Yaskawa INFORM job: A_ROOF_SIDE_0617_2_PAINT_48.JBI

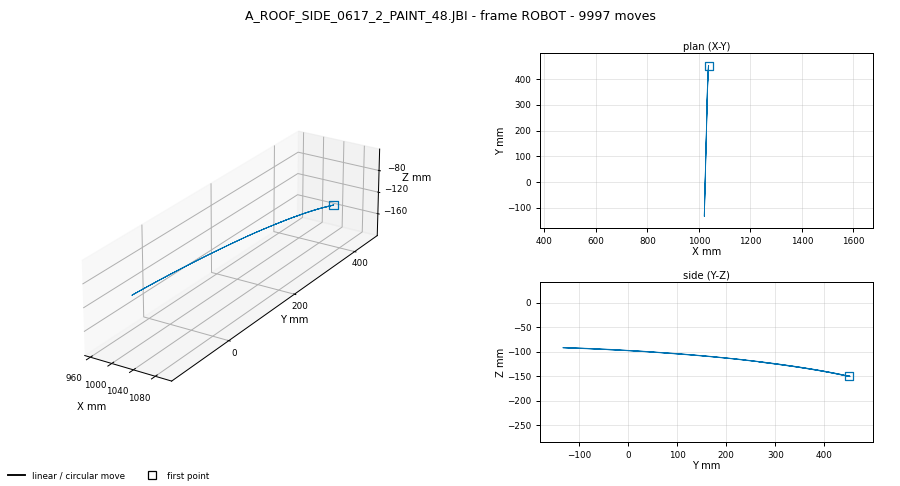
[picture p0: tool path of A_ROOF_SIDE_0617_2_PAINT_48.JBI in frame ROBOT, 9997 of 9997 moves have a stored position in this frame; points joined in program order, loops and branches not executed]
/JOB
//NAME A_ROOF_SIDE_0617_2_PAINT48
//POS
///NPOS 9997,0,0,0,0,0
///TOOL 1
///USER 0
///POSTYPE ROBOT
///RECTAN
///RCONF 1,0,0,0,0,0,0,0,0,0,0,0,0,0,0,0,0,0,0,0,0,0,0,0
C00000=1038.154,450.704,-149.023,176.566,47.258,159.897
C00001=1038.195,451.062,-149.082,176.595,47.266,159.904
C00002=1038.238,451.419,-149.141,176.623,47.275,159.910
C00003=1038.282,451.776,-149.199,176.652,47.283,159.916
C00004=1038.327,452.132,-149.255,176.680,47.290,159.922
C00005=1038.035,452.185,-149.577,176.684,47.363,159.945
C00006=1037.991,451.842,-149.523,176.655,47.356,159.939
C00007=1037.948,451.499,-149.468,176.628,47.348,159.933
C00008=1037.908,451.156,-149.412,176.601,47.340,159.927
C00009=1037.867,450.813,-149.355,176.574,47.332,159.921
C00010=1037.838,450.567,-149.314,176.554,47.326,159.916
C00011=1037.811,450.322,-149.271,176.535,47.321,159.912
C00012=1037.784,450.077,-149.230,176.516,47.315,159.908
C00013=1037.757,449.831,-149.186,176.496,47.309,159.904
C00014=1037.732,449.587,-149.144,176.477,47.303,159.899
C00015=1037.706,449.342,-149.100,176.459,47.296,159.895
C00016=1037.680,449.096,-149.056,176.440,47.290,159.890
C00017=1037.656,448.852,-149.011,176.421,47.283,159.886
C00018=1037.633,448.606,-148.966,176.403,47.277,159.882
C00019=1037.610,448.361,-148.921,176.384,47.271,159.877
C00020=1037.587,448.117,-148.875,176.366,47.263,159.873
C00021=1037.564,447.872,-148.829,176.348,47.257,159.868
C00022=1037.543,447.628,-148.782,176.328,47.250,159.864
C00023=1037.522,447.383,-148.734,176.310,47.243,159.859
C00024=1037.502,447.140,-148.687,176.292,47.236,159.855
C00025=1037.481,446.895,-148.639,176.274,47.229,159.850
C00026=1037.462,446.651,-148.590,176.256,47.221,159.846
C00027=1037.443,446.407,-148.542,176.237,47.214,159.841
C00028=1037.425,446.162,-148.492,176.220,47.207,159.837
C00029=1037.407,445.919,-148.443,176.203,47.199,159.832
C00030=1037.390,445.675,-148.391,176.184,47.192,159.828
C00031=1037.373,445.431,-148.341,176.167,47.184,159.823
C00032=1037.357,445.188,-148.290,176.149,47.177,159.818
C00033=1037.342,444.944,-148.238,176.132,47.169,159.814
C00034=1037.327,444.701,-148.186,176.115,47.161,159.809
C00035=1037.312,444.457,-148.134,176.098,47.153,159.805
C00036=1037.298,444.215,-148.081,176.080,47.145,159.800
C00037=1037.284,443.972,-148.027,176.063,47.136,159.795
C00038=1037.271,443.728,-147.974,176.046,47.128,159.790
C00039=1037.258,443.484,-147.920,176.029,47.120,159.786
C00040=1037.244,443.240,-147.867,176.013,47.112,159.781
C00041=1037.231,442.997,-147.814,175.995,47.104,159.777
C00042=1037.217,442.752,-147.761,175.979,47.096,159.772
C00043=1037.204,442.508,-147.708,175.962,47.087,159.768
C00044=1037.191,442.264,-147.654,175.945,47.080,159.763
C00045=1037.178,442.020,-147.601,175.928,47.072,159.759
C00046=1037.164,441.776,-147.549,175.912,47.063,159.754
C00047=1037.151,441.533,-147.495,175.895,47.055,159.750
C00048=1037.138,441.288,-147.443,175.879,47.047,159.745
C00049=1037.125,441.044,-147.390,175.862,47.040,159.741
C00050=1037.112,440.801,-147.337,175.845,47.032,159.736
C00051=1037.099,440.556,-147.285,175.829,47.024,159.732
C00052=1037.086,440.312,-147.232,175.813,47.016,159.728
C00053=1037.073,440.068,-147.179,175.798,47.008,159.723
C00054=1037.060,439.824,-147.126,175.782,47.000,159.719
C00055=1037.047,439.580,-147.075,175.766,46.993,159.715
C00056=1037.034,439.336,-147.022,175.749,46.985,159.710
C00057=1037.021,439.091,-146.970,175.733,46.977,159.706
C00058=1037.009,438.847,-146.917,175.717,46.970,159.702
C00059=1036.996,438.603,-146.866,175.701,46.962,159.697
C00060=1036.983,438.358,-146.813,175.686,46.954,159.693
C00061=1036.971,438.114,-146.761,175.670,46.946,159.689
C00062=1036.957,437.872,-146.709,175.654,46.939,159.685
C00063=1036.945,437.628,-146.657,175.639,46.931,159.681
C00064=1036.932,437.385,-146.606,175.624,46.924,159.677
C00065=1036.920,437.142,-146.553,175.609,46.916,159.672
C00066=1036.907,436.899,-146.502,175.593,46.909,159.668
C00067=1036.894,436.655,-146.450,175.578,46.901,159.664
C00068=1036.882,436.413,-146.399,175.562,46.894,159.660
C00069=1036.869,436.169,-146.348,175.548,46.886,159.656
C00070=1036.857,435.924,-146.296,175.532,46.879,159.652
C00071=1036.844,435.680,-146.245,175.517,46.871,159.648
C00072=1036.832,435.436,-146.193,175.502,46.864,159.644
C00073=1036.820,435.191,-146.142,175.487,46.857,159.640
C00074=1036.807,434.947,-146.091,175.472,46.849,159.636
C00075=1036.795,434.702,-146.039,175.457,46.842,159.632
C00076=1036.782,434.458,-145.988,175.442,46.835,159.628
C00077=1036.770,434.213,-145.937,175.427,46.828,159.624
C00078=1036.758,433.969,-145.886,175.413,46.821,159.620
C00079=1036.745,433.725,-145.835,175.398,46.813,159.616
C00080=1036.733,433.480,-145.784,175.384,46.806,159.612
C00081=1036.721,433.235,-145.734,175.369,46.799,159.609
C00082=1036.708,432.991,-145.683,175.354,46.792,159.605
C00083=1036.696,432.747,-145.632,175.340,46.785,159.601
C00084=1036.684,432.502,-145.581,175.325,46.778,159.597
C00085=1036.672,432.257,-145.530,175.311,46.771,159.593
C00086=1036.655,431.927,-145.462,175.292,46.762,159.588
C00087=1036.639,431.598,-145.394,175.272,46.752,159.583
C00088=1036.623,431.268,-145.327,175.253,46.742,159.578
C00089=1036.607,430.938,-145.258,175.234,46.733,159.573
C00090=1036.594,430.693,-145.208,175.220,46.726,159.569
C00091=1036.583,430.449,-145.158,175.207,46.719,159.566
C00092=1036.571,430.205,-145.107,175.193,46.712,159.562
C00093=1036.559,429.960,-145.057,175.178,46.706,159.558
C00094=1036.548,429.715,-145.006,175.164,46.699,159.555
C00095=1036.535,429.470,-144.956,175.151,46.692,159.551
C00096=1036.524,429.226,-144.906,175.137,46.685,159.547
C00097=1036.512,428.981,-144.856,175.123,46.678,159.544
C00098=1036.500,428.736,-144.806,175.110,46.671,159.540
C00099=1036.489,428.491,-144.756,175.096,46.665,159.537
C00100=1036.477,428.247,-144.706,175.083,46.658,159.533
C00101=1036.465,428.002,-144.657,175.069,46.651,159.529
C00102=1036.454,427.757,-144.607,175.055,46.645,159.526
C00103=1036.442,427.512,-144.557,175.042,46.638,159.522
C00104=1036.431,427.268,-144.508,175.028,46.631,159.519
C00105=1036.419,427.022,-144.458,175.015,46.625,159.515
C00106=1036.407,426.778,-144.409,175.002,46.618,159.512
C00107=1036.395,426.533,-144.359,174.988,46.612,159.509
C00108=1036.383,426.288,-144.310,174.976,46.605,159.505
C00109=1036.373,426.043,-144.260,174.962,46.599,159.502
C00110=1036.361,425.798,-144.211,174.949,46.592,159.498
C00111=1036.349,425.553,-144.162,174.936,46.586,159.495
C00112=1036.338,425.308,-144.113,174.922,46.579,159.491
C00113=1036.327,425.063,-144.064,174.910,46.573,159.488
C00114=1036.315,424.819,-144.015,174.897,46.566,159.485
C00115=1036.304,424.574,-143.966,174.884,46.560,159.481
C00116=1036.292,424.329,-143.917,174.871,46.554,159.478
C00117=1036.281,424.084,-143.868,174.858,46.548,159.475
C00118=1036.270,423.839,-143.818,174.845,46.541,159.471
C00119=1036.259,423.595,-143.769,174.833,46.535,159.468
C00120=1036.247,423.348,-143.721,174.820,46.528,159.465
C00121=1036.235,423.104,-143.672,174.807,46.522,159.461
C00122=1036.218,422.706,-143.593,174.787,46.512,159.456
C00123=1036.199,422.308,-143.515,174.767,46.502,159.451
C00124=1036.181,421.909,-143.436,174.747,46.492,159.446
C00125=1036.163,421.511,-143.357,174.726,46.482,159.441
C00126=1036.151,421.265,-143.309,174.714,46.476,159.437
C00127=1036.140,421.021,-143.261,174.702,46.470,159.434
C00128=1036.129,420.776,-143.212,174.689,46.464,159.431
C00129=1036.118,420.531,-143.164,174.677,46.458,159.428
C00130=1036.107,420.286,-143.116,174.664,46.452,159.425
C00131=1036.096,420.041,-143.068,174.653,46.446,159.422
C00132=1036.085,419.796,-143.020,174.641,46.440,159.419
C00133=1036.074,419.550,-142.971,174.628,46.434,159.416
C00134=1036.063,419.305,-142.925,174.616,46.428,159.413
C00135=1036.052,419.060,-142.876,174.604,46.423,159.410
C00136=1036.041,418.815,-142.828,174.593,46.417,159.407
C00137=1036.030,418.570,-142.780,174.580,46.411,159.403
C00138=1036.020,418.324,-142.733,174.568,46.405,159.400
C00139=1036.009,418.079,-142.685,174.557,46.399,159.397
C00140=1035.998,417.834,-142.636,174.545,46.393,159.394
C00141=1035.987,417.589,-142.590,174.533,46.388,159.391
C00142=1035.977,417.344,-142.542,174.521,46.382,159.388
C00143=1035.966,417.098,-142.494,174.509,46.376,159.385
C00144=1035.955,416.852,-142.447,174.498,46.370,159.383
C00145=1035.944,416.608,-142.399,174.486,46.365,159.380
C00146=1035.933,416.363,-142.352,174.475,46.359,159.377
C00147=1035.922,416.117,-142.305,174.463,46.353,159.374
C00148=1035.912,415.872,-142.258,174.452,46.348,159.371
C00149=1035.901,415.626,-142.210,174.440,46.342,159.368
C00150=1035.890,415.381,-142.164,174.429,46.337,159.365
C00151=1035.880,415.136,-142.116,174.417,46.331,159.362
C00152=1035.869,414.891,-142.069,174.406,46.325,159.359
C00153=1035.858,414.644,-142.022,174.394,46.320,159.357
C00154=1035.847,414.399,-141.976,174.383,46.314,159.354
C00155=1035.837,414.154,-141.928,174.372,46.309,159.351
C00156=1035.827,413.909,-141.881,174.360,46.303,159.348
C00157=1035.816,413.664,-141.835,174.349,46.298,159.345
C00158=1035.806,413.419,-141.787,174.339,46.292,159.342
C00159=1035.794,413.172,-141.741,174.327,46.287,159.340
C00160=1035.784,412.927,-141.694,174.316,46.281,159.337
C00161=1035.773,412.682,-141.647,174.305,46.276,159.334
C00162=1035.763,412.436,-141.601,174.294,46.271,159.331
C00163=1035.753,412.191,-141.554,174.282,46.265,159.329
C00164=1035.742,411.946,-141.507,174.272,46.260,159.326
C00165=1035.732,411.700,-141.460,174.261,46.254,159.323
C00166=1035.722,411.455,-141.415,174.250,46.249,159.320
C00167=1035.712,411.210,-141.368,174.239,46.244,159.318
C00168=1035.702,410.964,-141.322,174.229,46.239,159.315
C00169=1035.691,410.719,-141.276,174.218,46.233,159.312
C00170=1035.681,410.473,-141.229,174.206,46.228,159.310
C00171=1035.670,410.228,-141.183,174.196,46.223,159.307
C00172=1035.660,409.982,-141.137,174.185,46.218,159.304
C00173=1035.649,409.737,-141.091,174.174,46.213,159.302
C00174=1035.639,409.491,-141.044,174.164,46.208,159.299
C00175=1035.628,409.245,-140.998,174.153,46.203,159.297
C00176=1035.618,409.000,-140.953,174.143,46.197,159.294
C00177=1035.608,408.755,-140.907,174.132,46.192,159.291
C00178=1035.598,408.517,-140.863,174.122,46.188,159.289
C00179=1035.588,408.280,-140.819,174.112,46.182,159.286
C00180=1035.578,408.043,-140.775,174.102,46.177,159.284
C00181=1035.569,407.805,-140.730,174.091,46.173,159.281
C00182=1035.559,407.568,-140.686,174.082,46.168,159.279
C00183=1035.549,407.330,-140.642,174.072,46.163,159.277
C00184=1035.539,407.093,-140.598,174.061,46.159,159.274
C00185=1035.530,406.855,-140.554,174.052,46.153,159.272
C00186=1035.519,406.610,-140.508,174.041,46.148,159.269
C00187=1035.510,406.365,-140.462,174.031,46.144,159.267
C00188=1035.499,406.118,-140.417,174.021,46.139,159.264
C00189=1035.489,405.874,-140.371,174.010,46.134,159.262
C00190=1035.479,405.627,-140.326,174.001,46.129,159.259
C00191=1035.469,405.382,-140.281,173.990,46.124,159.257
C00192=1035.460,405.136,-140.235,173.980,46.119,159.254
C00193=1035.450,404.890,-140.190,173.970,46.114,159.252
C00194=1035.440,404.645,-140.145,173.960,46.110,159.249
C00195=1035.429,404.399,-140.099,173.950,46.104,159.247
C00196=1035.420,404.154,-140.054,173.940,46.100,159.244
C00197=1035.411,403.908,-140.009,173.929,46.095,159.242
C00198=1035.400,403.662,-139.964,173.920,46.090,159.240
C00199=1035.391,403.416,-139.919,173.910,46.086,159.237
C00200=1035.381,403.171,-139.873,173.900,46.081,159.235
C00201=1035.371,402.926,-139.828,173.890,46.076,159.233
C00202=1035.361,402.679,-139.783,173.880,46.072,159.230
C00203=1035.352,402.433,-139.739,173.871,46.067,159.228
C00204=1035.342,402.188,-139.694,173.861,46.062,159.225
C00205=1035.333,401.942,-139.649,173.851,46.058,159.223
C00206=1035.323,401.697,-139.604,173.841,46.053,159.221
C00207=1035.313,401.450,-139.559,173.831,46.049,159.218
C00208=1035.303,401.205,-139.514,173.822,46.044,159.216
C00209=1035.293,400.959,-139.470,173.812,46.039,159.214
C00210=1035.284,400.713,-139.425,173.802,46.034,159.211
C00211=1035.274,400.468,-139.380,173.792,46.030,159.209
C00212=1035.264,400.222,-139.337,173.783,46.026,159.207
C00213=1035.254,399.976,-139.292,173.773,46.021,159.205
C00214=1035.245,399.730,-139.248,173.764,46.017,159.202
C00215=1035.235,399.485,-139.203,173.755,46.012,159.200
C00216=1035.226,399.239,-139.159,173.745,46.008,159.198
C00217=1035.216,398.993,-139.114,173.736,46.003,159.196
C00218=1035.207,398.747,-139.070,173.726,45.999,159.193
C00219=1035.196,398.501,-139.026,173.717,45.994,159.191
C00220=1035.187,398.255,-138.982,173.707,45.990,159.189
C00221=1035.177,398.010,-138.938,173.698,45.986,159.187
C00222=1035.168,397.764,-138.894,173.689,45.981,159.185
C00223=1035.158,397.518,-138.850,173.679,45.977,159.182
C00224=1035.149,397.272,-138.806,173.670,45.973,159.180
C00225=1035.139,397.026,-138.762,173.661,45.969,159.178
C00226=1035.130,396.780,-138.718,173.651,45.964,159.176
C00227=1035.120,396.535,-138.675,173.642,45.960,159.174
C00228=1035.111,396.289,-138.631,173.633,45.956,159.172
C00229=1035.102,396.042,-138.587,173.624,45.951,159.169
C00230=1035.092,395.796,-138.542,173.614,45.947,159.167
C00231=1035.083,395.551,-138.499,173.605,45.943,159.165
C00232=1035.073,395.305,-138.455,173.596,45.939,159.163
C00233=1035.064,395.059,-138.411,173.588,45.934,159.161
C00234=1035.055,394.814,-138.367,173.578,45.930,159.159
C00235=1035.045,394.568,-138.324,173.569,45.927,159.157
C00236=1035.036,394.321,-138.280,173.560,45.922,159.155
C00237=1035.026,394.076,-138.237,173.551,45.918,159.153
C00238=1035.018,393.848,-138.196,173.543,45.914,159.151
C00239=1035.010,393.621,-138.157,173.535,45.910,159.149
C00240=1035.001,393.394,-138.117,173.527,45.907,159.147
C00241=1034.992,393.167,-138.077,173.518,45.903,159.145
C00242=1034.983,392.940,-138.037,173.510,45.899,159.143
C00243=1034.976,392.712,-137.997,173.502,45.896,159.141
C00244=1034.966,392.485,-137.957,173.493,45.892,159.139
C00245=1034.958,392.258,-137.917,173.486,45.888,159.138
C00246=1034.948,392.012,-137.874,173.477,45.884,159.135
C00247=1034.940,391.766,-137.831,173.467,45.880,159.133
C00248=1034.930,391.520,-137.787,173.459,45.877,159.132
C00249=1034.921,391.274,-137.744,173.450,45.872,159.129
C00250=1034.912,391.028,-137.701,173.441,45.869,159.127
C00251=1034.903,390.782,-137.659,173.433,45.865,159.126
C00252=1034.894,390.536,-137.615,173.424,45.861,159.123
C00253=1034.884,390.290,-137.572,173.415,45.857,159.122
C00254=1034.875,390.044,-137.529,173.407,45.853,159.120
C00255=1034.866,389.798,-137.487,173.398,45.849,159.118
C00256=1034.856,389.551,-137.444,173.390,45.846,159.116
C00257=1034.848,389.305,-137.401,173.381,45.841,159.114
C00258=1034.839,389.060,-137.358,173.373,45.837,159.112
C00259=1034.829,388.814,-137.316,173.365,45.833,159.110
C00260=1034.821,388.567,-137.273,173.356,45.830,159.108
C00261=1034.811,388.321,-137.231,173.347,45.826,159.106
C00262=1034.803,388.075,-137.188,173.339,45.822,159.104
C00263=1034.794,387.829,-137.145,173.331,45.819,159.102
C00264=1034.784,387.583,-137.103,173.322,45.815,159.100
C00265=1034.776,387.336,-137.060,173.313,45.812,159.099
C00266=1034.766,387.090,-137.018,173.305,45.808,159.097
C00267=1034.757,386.844,-136.975,173.297,45.804,159.095
C00268=1034.748,386.598,-136.934,173.289,45.801,159.093
C00269=1034.739,386.352,-136.891,173.280,45.797,159.091
C00270=1034.729,386.105,-136.849,173.272,45.793,159.089
C00271=1034.720,385.860,-136.807,173.264,45.790,159.087
C00272=1034.712,385.613,-136.764,173.255,45.786,159.086
C00273=1034.703,385.366,-136.723,173.248,45.783,159.084
C00274=1034.694,385.121,-136.680,173.239,45.779,159.082
C00275=1034.685,384.874,-136.638,173.231,45.776,159.080
C00276=1034.676,384.628,-136.597,173.222,45.772,159.078
C00277=1034.667,384.382,-136.554,173.214,45.769,159.077
C00278=1034.658,384.136,-136.513,173.206,45.765,159.075
C00279=1034.649,383.890,-136.471,173.198,45.761,159.073
C00280=1034.641,383.643,-136.429,173.190,45.758,159.071
C00281=1034.631,383.397,-136.386,173.182,45.754,159.069
C00282=1034.622,383.151,-136.344,173.174,45.751,159.068
C00283=1034.614,382.904,-136.303,173.166,45.748,159.066
C00284=1034.605,382.658,-136.261,173.158,45.744,159.064
C00285=1034.596,382.412,-136.219,173.150,45.740,159.062
C00286=1034.587,382.166,-136.178,173.142,45.737,159.061
C00287=1034.578,381.920,-136.136,173.134,45.734,159.059
C00288=1034.569,381.673,-136.094,173.126,45.730,159.057
C00289=1034.561,381.427,-136.053,173.118,45.727,159.055
C00290=1034.552,381.180,-136.010,173.110,45.723,159.054
C00291=1034.543,380.934,-135.969,173.102,45.720,159.052
C00292=1034.535,380.688,-135.928,173.095,45.716,159.050
C00293=1034.526,380.441,-135.886,173.087,45.713,159.048
C00294=1034.518,380.195,-135.845,173.078,45.710,159.047
C00295=1034.509,379.948,-135.803,173.071,45.707,159.045
C00296=1034.500,379.703,-135.762,173.063,45.703,159.043
C00297=1034.492,379.456,-135.721,173.055,45.700,159.042
C00298=1034.484,379.246,-135.685,173.049,45.698,159.040
C00299=1034.477,379.037,-135.650,173.042,45.695,159.039
C00300=1034.470,378.826,-135.614,173.036,45.691,159.037
C00301=1034.463,378.617,-135.580,173.029,45.689,159.036
C00302=1034.455,378.407,-135.544,173.022,45.686,159.035
C00303=1034.448,378.198,-135.509,173.016,45.683,159.033
C00304=1034.441,377.988,-135.474,173.009,45.681,159.032
C00305=1034.434,377.778,-135.440,173.002,45.678,159.030
C00306=1034.425,377.532,-135.398,172.996,45.675,159.029
C00307=1034.416,377.285,-135.357,172.987,45.672,159.027
C00308=1034.408,377.038,-135.316,172.980,45.669,159.026
C00309=1034.398,376.792,-135.275,172.972,45.666,159.024
C00310=1034.390,376.545,-135.234,172.965,45.663,159.022
C00311=1034.382,376.299,-135.194,172.957,45.659,159.021
C00312=1034.373,376.052,-135.153,172.950,45.657,159.019
C00313=1034.364,375.806,-135.112,172.943,45.653,159.018
C00314=1034.355,375.560,-135.071,172.935,45.650,159.016
C00315=1034.347,375.313,-135.030,172.927,45.647,159.014
C00316=1034.339,375.066,-134.989,172.919,45.644,159.013
C00317=1034.330,374.820,-134.949,172.912,45.641,159.011
C00318=1034.321,374.573,-134.908,172.905,45.638,159.010
C00319=1034.313,374.327,-134.867,172.897,45.635,159.008
C00320=1034.305,374.080,-134.826,172.890,45.632,159.007
C00321=1034.296,373.834,-134.786,172.882,45.629,159.005
C00322=1034.288,373.588,-134.746,172.875,45.626,159.003
C00323=1034.279,373.341,-134.705,172.868,45.623,159.002
C00324=1034.270,373.095,-134.665,172.860,45.620,159.000
C00325=1034.262,372.849,-134.624,172.853,45.617,158.999
C00326=1034.254,372.601,-134.584,172.846,45.614,158.997
C00327=1034.246,372.355,-134.543,172.839,45.612,158.996
C00328=1034.237,372.109,-134.503,172.831,45.609,158.994
C00329=1034.229,371.862,-134.462,172.824,45.606,158.993
C00330=1034.221,371.615,-134.422,172.817,45.603,158.991
C00331=1034.213,371.369,-134.382,172.810,45.600,158.990
C00332=1034.204,371.123,-134.342,172.802,45.597,158.988
C00333=1034.196,370.875,-134.301,172.795,45.594,158.987
C00334=1034.188,370.629,-134.261,172.788,45.591,158.985
C00335=1034.179,370.383,-134.221,172.781,45.588,158.984
C00336=1034.171,370.136,-134.181,172.773,45.586,158.982
C00337=1034.163,369.890,-134.140,172.766,45.583,158.981
C00338=1034.154,369.642,-134.100,172.759,45.580,158.979
C00339=1034.146,369.396,-134.060,172.753,45.577,158.978
C00340=1034.138,369.149,-134.020,172.746,45.575,158.977
C00341=1034.130,368.903,-133.980,172.738,45.572,158.975
C00342=1034.121,368.657,-133.940,172.731,45.569,158.974
C00343=1034.112,368.409,-133.901,172.724,45.567,158.972
C00344=1034.105,368.162,-133.861,172.717,45.564,158.971
C00345=1034.096,367.916,-133.822,172.711,45.561,158.970
C00346=1034.088,367.669,-133.782,172.703,45.559,158.968
C00347=1034.080,367.423,-133.742,172.696,45.556,158.967
C00348=1034.071,367.176,-133.702,172.689,45.553,158.965
C00349=1034.063,366.929,-133.662,172.682,45.550,158.964
C00350=1034.055,366.683,-133.623,172.675,45.548,158.962
C00351=1034.047,366.436,-133.583,172.668,45.545,158.961
C00352=1034.039,366.189,-133.544,172.662,45.543,158.960
C00353=1034.030,365.943,-133.504,172.655,45.540,158.958
C00354=1034.023,365.696,-133.464,172.648,45.537,158.957
C00355=1034.014,365.449,-133.425,172.640,45.535,158.956
C00356=1034.006,365.203,-133.386,172.633,45.532,158.954
C00357=1033.998,364.956,-133.346,172.627,45.530,158.953
C00358=1033.985,364.557,-133.283,172.616,45.526,158.951
C00359=1033.972,364.158,-133.219,172.605,45.522,158.948
C00360=1033.958,363.759,-133.155,172.594,45.518,158.946
C00361=1033.945,363.361,-133.092,172.584,45.514,158.944
C00362=1033.938,363.114,-133.052,172.577,45.511,158.943
C00363=1033.929,362.867,-133.013,172.570,45.508,158.941
C00364=1033.921,362.620,-132.974,172.563,45.506,158.940
C00365=1033.913,362.373,-132.934,172.557,45.503,158.939
C00366=1033.905,362.126,-132.895,172.550,45.501,158.938
C00367=1033.898,361.879,-132.856,172.543,45.499,158.936
C00368=1033.890,361.633,-132.817,172.537,45.496,158.935
C00369=1033.882,361.386,-132.778,172.530,45.494,158.934
C00370=1033.873,361.139,-132.739,172.523,45.492,158.932
C00371=1033.865,360.892,-132.700,172.517,45.489,158.931
C00372=1033.858,360.646,-132.660,172.510,45.487,158.930
C00373=1033.850,360.398,-132.622,172.503,45.484,158.928
C00374=1033.841,360.152,-132.583,172.497,45.482,158.927
C00375=1033.833,359.905,-132.544,172.490,45.480,158.926
C00376=1033.826,359.658,-132.506,172.483,45.477,158.925
C00377=1033.817,359.412,-132.466,172.478,45.475,158.923
C00378=1033.809,359.164,-132.428,172.471,45.473,158.922
C00379=1033.801,358.918,-132.390,172.465,45.470,158.921
C00380=1033.793,358.671,-132.351,172.458,45.468,158.920
C00381=1033.785,358.423,-132.312,172.451,45.466,158.918
C00382=1033.777,358.177,-132.273,172.445,45.464,158.917
C00383=1033.769,357.930,-132.235,172.438,45.461,158.916
C00384=1033.761,357.683,-132.196,172.432,45.459,158.915
C00385=1033.753,357.437,-132.158,172.425,45.457,158.913
C00386=1033.745,357.189,-132.119,172.419,45.454,158.912
C00387=1033.738,356.943,-132.081,172.413,45.453,158.911
C00388=1033.729,356.696,-132.042,172.406,45.450,158.910
C00389=1033.721,356.448,-132.004,172.400,45.448,158.909
C00390=1033.714,356.202,-131.966,172.393,45.446,158.907
C00391=1033.706,355.954,-131.926,172.388,45.443,158.906
C00392=1033.699,355.708,-131.888,172.381,45.442,158.905
C00393=1033.690,355.461,-131.850,172.375,45.440,158.904
C00394=1033.682,355.214,-131.812,172.368,45.437,158.903
C00395=1033.675,354.967,-131.774,172.362,45.436,158.902
C00396=1033.667,354.720,-131.736,172.356,45.433,158.900
C00397=1033.659,354.473,-131.697,172.350,45.431,158.899
C00398=1033.651,354.226,-131.659,172.343,45.429,158.898
C00399=1033.643,353.979,-131.622,172.337,45.427,158.897
C00400=1033.635,353.732,-131.583,172.330,45.425,158.896
C00401=1033.627,353.485,-131.545,172.325,45.423,158.895
C00402=1033.620,353.238,-131.507,172.318,45.420,158.893
C00403=1033.612,352.991,-131.469,172.312,45.419,158.892
C00404=1033.603,352.744,-131.431,172.306,45.417,158.891
C00405=1033.596,352.497,-131.393,172.300,45.415,158.890
C00406=1033.588,352.250,-131.355,172.293,45.412,158.889
C00407=1033.581,352.003,-131.317,172.287,45.411,158.888
C00408=1033.573,351.756,-131.279,172.282,45.408,158.886
C00409=1033.565,351.509,-131.241,172.275,45.407,158.885
C00410=1033.557,351.262,-131.203,172.269,45.405,158.884
C00411=1033.550,351.015,-131.166,172.264,45.403,158.883
C00412=1033.542,350.768,-131.127,172.257,45.401,158.882
C00413=1033.534,350.521,-131.090,172.251,45.399,158.881
C00414=1033.522,350.128,-131.030,172.242,45.396,158.879
C00415=1033.510,349.736,-130.970,172.231,45.393,158.877
C00416=1033.498,349.343,-130.910,172.222,45.390,158.876
C00417=1033.485,348.951,-130.850,172.213,45.387,158.874
C00418=1033.478,348.703,-130.813,172.207,45.385,158.873
C00419=1033.470,348.457,-130.776,172.200,45.383,158.872
C00420=1033.463,348.209,-130.738,172.195,45.381,158.871
C00421=1033.454,347.963,-130.700,172.188,45.379,158.870
C00422=1033.447,347.715,-130.663,172.182,45.377,158.868
C00423=1033.439,347.468,-130.625,172.177,45.376,158.868
C00424=1033.431,347.221,-130.588,172.171,45.374,158.866
C00425=1033.424,346.974,-130.551,172.165,45.372,158.865
C00426=1033.416,346.727,-130.514,172.159,45.370,158.864
C00427=1033.408,346.480,-130.476,172.153,45.369,158.863
C00428=1033.400,346.233,-130.439,172.147,45.367,158.862
C00429=1033.393,345.986,-130.402,172.141,45.365,158.861
C00430=1033.385,345.739,-130.365,172.136,45.363,158.860
C00431=1033.378,345.491,-130.328,172.129,45.362,158.859
C00432=1033.370,345.244,-130.291,172.124,45.359,158.858
C00433=1033.363,344.997,-130.253,172.118,45.358,158.857
C00434=1033.356,344.750,-130.216,172.113,45.356,158.856
C00435=1033.348,344.503,-130.179,172.106,45.354,158.855
C00436=1033.340,344.256,-130.142,172.101,45.353,158.854
C00437=1033.333,344.009,-130.105,172.095,45.351,158.853
C00438=1033.325,343.762,-130.068,172.089,45.350,158.852
C00439=1033.318,343.515,-130.031,172.083,45.348,158.851
C00440=1033.310,343.267,-129.994,172.077,45.346,158.850
C00441=1033.303,343.020,-129.957,172.072,45.344,158.849
C00442=1033.295,342.773,-129.920,172.066,45.343,158.848
C00443=1033.288,342.525,-129.883,172.060,45.341,158.847
C00444=1033.280,342.279,-129.846,172.054,45.340,158.846
C00445=1033.273,342.031,-129.809,172.049,45.338,158.845
C00446=1033.265,341.784,-129.773,172.044,45.336,158.844
C00447=1033.257,341.537,-129.736,172.038,45.335,158.843
C00448=1033.250,341.289,-129.699,172.032,45.333,158.842
C00449=1033.242,341.043,-129.662,172.026,45.331,158.841
C00450=1033.235,340.795,-129.625,172.021,45.329,158.840
C00451=1033.227,340.547,-129.589,172.015,45.328,158.839
C00452=1033.219,340.301,-129.552,172.009,45.327,158.838
C00453=1033.212,340.054,-129.516,172.003,45.325,158.837
C00454=1033.205,339.806,-129.480,171.998,45.323,158.836
C00455=1033.197,339.559,-129.442,171.992,45.322,158.835
C00456=1033.190,339.312,-129.406,171.987,45.321,158.834
C00457=1033.182,339.064,-129.370,171.982,45.319,158.834
C00458=1033.174,338.818,-129.333,171.976,45.318,158.833
C00459=1033.166,338.570,-129.297,171.970,45.316,158.832
C00460=1033.160,338.323,-129.260,171.964,45.315,158.831
C00461=1033.152,338.076,-129.224,171.959,45.313,158.830
C00462=1033.145,337.828,-129.188,171.953,45.312,158.829
C00463=1033.137,337.581,-129.152,171.948,45.310,158.828
C00464=1033.129,337.334,-129.115,171.943,45.309,158.827
C00465=1033.122,337.087,-129.079,171.937,45.307,158.826
C00466=1033.115,336.839,-129.042,171.931,45.306,158.825
C00467=1033.107,336.592,-129.006,171.926,45.304,158.824
C00468=1033.100,336.345,-128.970,171.920,45.303,158.823
C00469=1033.093,336.098,-128.934,171.915,45.302,158.823
C00470=1033.081,335.702,-128.875,171.907,45.300,158.821
C00471=1033.070,335.306,-128.818,171.898,45.297,158.820
C00472=1033.057,334.910,-128.760,171.889,45.295,158.818
C00473=1033.045,334.513,-128.702,171.880,45.293,158.817
C00474=1033.038,334.267,-128.666,171.875,45.291,158.816
C00475=1033.030,334.019,-128.630,171.869,45.290,158.815
C00476=1033.023,333.772,-128.594,171.864,45.289,158.814
C00477=1033.016,333.524,-128.559,171.859,45.287,158.813
C00478=1033.008,333.277,-128.523,171.853,45.287,158.812
C00479=1033.001,333.030,-128.487,171.848,45.285,158.812
C00480=1032.994,332.782,-128.451,171.843,45.284,158.811
C00481=1032.986,332.535,-128.415,171.838,45.282,158.810
C00482=1032.979,332.288,-128.379,171.832,45.281,158.809
C00483=1032.972,332.040,-128.344,171.827,45.280,158.808
C00484=1032.964,331.793,-128.308,171.822,45.278,158.807
C00485=1032.956,331.546,-128.272,171.816,45.278,158.807
C00486=1032.950,331.299,-128.237,171.811,45.276,158.806
C00487=1032.942,331.051,-128.201,171.806,45.275,158.805
C00488=1032.935,330.804,-128.166,171.801,45.274,158.804
C00489=1032.927,330.556,-128.129,171.795,45.272,158.803
C00490=1032.921,330.309,-128.094,171.790,45.271,158.802
C00491=1032.913,330.062,-128.058,171.785,45.270,158.802
C00492=1032.906,329.814,-128.023,171.780,45.269,158.801
C00493=1032.899,329.567,-127.987,171.774,45.268,158.800
C00494=1032.891,329.320,-127.952,171.769,45.266,158.799
C00495=1032.883,329.072,-127.916,171.764,45.265,158.798
C00496=1032.877,328.825,-127.881,171.759,45.264,158.797
C00497=1032.869,328.578,-127.845,171.753,45.263,158.797
C00498=1032.862,328.330,-127.810,171.748,45.262,158.796
C00499=1032.855,328.083,-127.774,171.743,45.261,158.795
C00500=1032.847,327.835,-127.739,171.738,45.259,158.794
C00501=1032.840,327.588,-127.704,171.733,45.258,158.793
C00502=1032.832,327.340,-127.669,171.727,45.258,158.793
C00503=1032.825,327.093,-127.634,171.722,45.256,158.792
C00504=1032.818,326.846,-127.599,171.717,45.255,158.791
C00505=1032.810,326.598,-127.564,171.713,45.254,158.790
C00506=1032.803,326.351,-127.529,171.706,45.253,158.789
C00507=1032.796,326.103,-127.493,171.702,45.252,158.789
C00508=1032.788,325.856,-127.459,171.697,45.251,158.788
C00509=1032.781,325.608,-127.424,171.692,45.250,158.787
C00510=1032.773,325.361,-127.389,171.687,45.249,158.786
C00511=1032.766,325.113,-127.354,171.681,45.248,158.786
C00512=1032.759,324.866,-127.319,171.676,45.247,158.785
C00513=1032.752,324.618,-127.284,171.671,45.246,158.784
C00514=1032.744,324.371,-127.249,171.667,45.245,158.784
C00515=1032.737,324.124,-127.214,171.662,45.245,158.783
C00516=1032.729,323.876,-127.179,171.657,45.243,158.782
C00517=1032.722,323.629,-127.145,171.651,45.242,158.781
C00518=1032.715,323.382,-127.109,171.646,45.241,158.780
C00519=1032.707,323.135,-127.075,171.641,45.241,158.780
C00520=1032.700,322.886,-127.039,171.636,45.240,158.779
C00521=1032.693,322.639,-127.006,171.632,45.239,158.778
C00522=1032.686,322.391,-126.970,171.627,45.238,158.778
C00523=1032.679,322.144,-126.936,171.622,45.237,158.777
C00524=1032.671,321.896,-126.900,171.616,45.236,158.776
C00525=1032.664,321.649,-126.866,171.611,45.235,158.775
C00526=1032.652,321.249,-126.810,171.604,45.234,158.774
C00527=1032.640,320.848,-126.755,171.595,45.232,158.773
C00528=1032.629,320.447,-126.697,171.587,45.231,158.772
C00529=1032.618,320.047,-126.642,171.580,45.229,158.771
C00530=1032.610,319.800,-126.607,171.575,45.228,158.770
C00531=1032.604,319.552,-126.573,171.570,45.227,158.769
C00532=1032.596,319.305,-126.539,171.565,45.226,158.769
C00533=1032.589,319.056,-126.504,171.560,45.225,158.768
C00534=1032.582,318.809,-126.469,171.555,45.225,158.767
C00535=1032.574,318.562,-126.435,171.550,45.224,158.767
C00536=1032.568,318.314,-126.400,171.545,45.223,158.766
C00537=1032.560,318.067,-126.366,171.540,45.223,158.765
C00538=1032.554,317.819,-126.331,171.535,45.222,158.764
C00539=1032.546,317.572,-126.297,171.531,45.221,158.764
C00540=1032.539,317.324,-126.263,171.526,45.220,158.763
C00541=1032.532,317.077,-126.228,171.521,45.219,158.762
C00542=1032.525,316.829,-126.194,171.516,45.219,158.762
C00543=1032.518,316.581,-126.160,171.512,45.218,158.761
C00544=1032.511,316.334,-126.125,171.507,45.217,158.760
C00545=1032.504,316.086,-126.091,171.502,45.216,158.760
C00546=1032.497,315.839,-126.056,171.497,45.215,158.759
C00547=1032.490,315.592,-126.023,171.493,45.215,158.758
C00548=1032.484,315.344,-125.988,171.488,45.214,158.758
C00549=1032.476,315.097,-125.954,171.483,45.213,158.757
C00550=1032.469,314.850,-125.920,171.478,45.212,158.756
C00551=1032.463,314.602,-125.885,171.474,45.211,158.756
C00552=1032.455,314.355,-125.851,171.469,45.210,158.755
C00553=1032.449,314.107,-125.816,171.464,45.210,158.754
C00554=1032.442,313.859,-125.783,171.459,45.209,158.754
C00555=1032.435,313.612,-125.749,171.454,45.208,158.753
C00556=1032.428,313.365,-125.714,171.451,45.207,158.752
C00557=1032.421,313.117,-125.680,171.446,45.206,158.752
C00558=1032.415,312.869,-125.646,171.441,45.206,158.751
C00559=1032.407,312.621,-125.612,171.436,45.205,158.750
C00560=1032.401,312.374,-125.578,171.432,45.204,158.750
C00561=1032.394,312.126,-125.544,171.427,45.204,158.749
C00562=1032.387,311.879,-125.510,171.422,45.203,158.748
C00563=1032.380,311.632,-125.476,171.417,45.202,158.748
C00564=1032.373,311.384,-125.441,171.413,45.202,158.747
C00565=1032.367,311.137,-125.408,171.408,45.201,158.746
C00566=1032.359,310.889,-125.375,171.403,45.200,158.746
C00567=1032.352,310.641,-125.341,171.399,45.200,158.745
C00568=1032.344,310.393,-125.308,171.394,45.199,158.745
C00569=1032.337,310.146,-125.274,171.390,45.199,158.744
C00570=1032.329,309.898,-125.241,171.385,45.198,158.744
C00571=1032.323,309.651,-125.207,171.380,45.198,158.743
C00572=1032.316,309.403,-125.174,171.376,45.197,158.742
C00573=1032.309,309.155,-125.140,171.371,45.197,158.742
C00574=1032.301,308.908,-125.106,171.366,45.196,158.741
C00575=1032.294,308.661,-125.074,171.363,45.195,158.741
C00576=1032.287,308.413,-125.040,171.358,45.195,158.740
C00577=1032.280,308.165,-125.007,171.353,45.195,158.740
C00578=1032.273,307.917,-124.973,171.349,45.194,158.739
C00579=1032.266,307.670,-124.941,171.344,45.194,158.738
C00580=1032.259,307.422,-124.907,171.340,45.193,158.738
C00581=1032.251,307.175,-124.873,171.335,45.193,158.737
C00582=1032.240,306.779,-124.820,171.328,45.192,158.736
C00583=1032.229,306.383,-124.767,171.321,45.191,158.735
C00584=1032.218,305.988,-124.714,171.313,45.190,158.734
C00585=1032.207,305.592,-124.661,171.306,45.190,158.734
C00586=1032.199,305.344,-124.628,171.302,45.190,158.733
C00587=1032.193,305.097,-124.595,171.297,45.189,158.732
C00588=1032.186,304.849,-124.561,171.293,45.188,158.732
C00589=1032.179,304.601,-124.528,171.289,45.188,158.731
C00590=1032.171,304.354,-124.495,171.284,45.188,158.731
C00591=1032.164,304.106,-124.462,171.279,45.187,158.730
C00592=1032.158,303.859,-124.429,171.275,45.187,158.730
C00593=1032.151,303.611,-124.396,171.270,45.187,158.729
C00594=1032.143,303.363,-124.362,171.266,45.186,158.729
C00595=1032.137,303.116,-124.330,171.262,45.186,158.728
C00596=1032.130,302.867,-124.297,171.257,45.185,158.727
C00597=1032.123,302.620,-124.263,171.253,45.184,158.727
C00598=1032.116,302.372,-124.231,171.248,45.184,158.726
C00599=1032.109,302.125,-124.198,171.244,45.184,158.726
C00600=1032.102,301.877,-124.164,171.239,45.183,158.725
C00601=1032.096,301.630,-124.131,171.236,45.183,158.725
C00602=1032.088,301.382,-124.099,171.231,45.183,158.724
C00603=1032.082,301.134,-124.066,171.226,45.182,158.724
C00604=1032.075,300.886,-124.032,171.222,45.182,158.723
C00605=1032.068,300.639,-124.000,171.217,45.182,158.723
C00606=1032.061,300.391,-123.967,171.214,45.181,158.722
C00607=1032.054,300.143,-123.934,171.209,45.181,158.721
C00608=1032.047,299.896,-123.900,171.205,45.180,158.721
C00609=1032.040,299.648,-123.868,171.200,45.180,158.720
C00610=1032.034,299.401,-123.835,171.197,45.180,158.720
C00611=1032.027,299.152,-123.802,171.192,45.179,158.719
C00612=1032.020,298.905,-123.770,171.188,45.179,158.719
C00613=1032.013,298.657,-123.737,171.183,45.179,158.718
C00614=1032.007,298.409,-123.704,171.180,45.179,158.718
C00615=1032.000,298.162,-123.672,171.175,45.178,158.717
C00616=1031.993,297.914,-123.639,171.170,45.178,158.717
C00617=1031.986,297.667,-123.606,171.166,45.178,158.716
C00618=1031.980,297.419,-123.573,171.162,45.177,158.716
C00619=1031.972,297.171,-123.540,171.158,45.177,158.715
C00620=1031.966,296.923,-123.508,171.153,45.176,158.715
C00621=1031.960,296.676,-123.475,171.150,45.176,158.714
C00622=1031.952,296.428,-123.442,171.145,45.176,158.714
C00623=1031.946,296.180,-123.410,171.141,45.176,158.713
C00624=1031.940,295.932,-123.378,171.136,45.175,158.713
C00625=1031.933,295.684,-123.344,171.133,45.175,158.712
C00626=1031.926,295.436,-123.312,171.128,45.175,158.712
C00627=1031.920,295.189,-123.280,171.124,45.174,158.711
C00628=1031.913,294.941,-123.247,171.120,45.174,158.711
C00629=1031.906,294.693,-123.214,171.116,45.174,158.710
C00630=1031.899,294.446,-123.182,171.111,45.174,158.710
C00631=1031.892,294.198,-123.149,171.108,45.174,158.710
C00632=1031.886,293.950,-123.117,171.103,45.173,158.709
C00633=1031.879,293.702,-123.085,171.099,45.173,158.708
C00634=1031.872,293.455,-123.053,171.094,45.173,158.708
C00635=1031.866,293.207,-123.021,171.091,45.173,158.708
C00636=1031.858,292.959,-122.988,171.086,45.172,158.707
C00637=1031.851,292.712,-122.956,171.082,45.173,158.707
C00638=1031.841,292.332,-122.907,171.076,45.172,158.706
C00639=1031.830,291.954,-122.858,171.070,45.172,158.705
C00640=1031.820,291.576,-122.809,171.063,45.172,158.705
C00641=1031.809,291.197,-122.760,171.057,45.172,158.704
C00642=1031.803,290.949,-122.728,171.053,45.172,158.703
C00643=1031.796,290.701,-122.695,171.048,45.172,158.703
C00644=1031.789,290.453,-122.664,171.045,45.172,158.703
C00645=1031.782,290.205,-122.632,171.040,45.171,158.702
C00646=1031.775,289.958,-122.600,171.036,45.172,158.702
C00647=1031.769,289.710,-122.568,171.033,45.171,158.701
C00648=1031.762,289.462,-122.536,171.028,45.171,158.701
C00649=1031.755,289.214,-122.504,171.024,45.171,158.700
C00650=1031.748,288.966,-122.472,171.020,45.171,158.700
C00651=1031.742,288.718,-122.440,171.016,45.171,158.700
C00652=1031.735,288.470,-122.409,171.012,45.171,158.699
C00653=1031.728,288.223,-122.376,171.008,45.171,158.699
C00654=1031.721,287.975,-122.345,171.004,45.171,158.698
C00655=1031.714,287.726,-122.313,170.999,45.171,158.698
C00656=1031.707,287.479,-122.281,170.996,45.171,158.697
C00657=1031.700,287.231,-122.250,170.992,45.171,158.697
C00658=1031.694,286.983,-122.218,170.988,45.171,158.697
C00659=1031.687,286.735,-122.186,170.984,45.170,158.696
C00660=1031.680,286.488,-122.154,170.979,45.171,158.696
C00661=1031.674,286.240,-122.123,170.976,45.171,158.695
C00662=1031.667,285.992,-122.091,170.972,45.171,158.695
C00663=1031.660,285.744,-122.060,170.967,45.171,158.694
C00664=1031.653,285.496,-122.028,170.964,45.171,158.694
C00665=1031.646,285.248,-121.997,170.960,45.171,158.694
C00666=1031.639,285.000,-121.964,170.956,45.171,158.693
C00667=1031.632,284.752,-121.933,170.952,45.171,158.693
C00668=1031.626,284.505,-121.902,170.947,45.171,158.693
C00669=1031.619,284.257,-121.870,170.944,45.171,158.692
C00670=1031.612,284.009,-121.839,170.940,45.171,158.692
C00671=1031.605,283.761,-121.808,170.936,45.172,158.691
C00672=1031.598,283.513,-121.776,170.932,45.171,158.691
C00673=1031.591,283.265,-121.745,170.928,45.171,158.691
C00674=1031.585,283.017,-121.714,170.924,45.171,158.690
C00675=1031.578,282.770,-121.682,170.920,45.172,158.690
C00676=1031.571,282.522,-121.651,170.916,45.172,158.689
C00677=1031.564,282.274,-121.619,170.912,45.171,158.689
C00678=1031.558,282.026,-121.588,170.908,45.172,158.689
C00679=1031.551,281.777,-121.557,170.905,45.172,158.688
C00680=1031.545,281.529,-121.526,170.900,45.172,158.688
C00681=1031.538,281.282,-121.494,170.897,45.172,158.688
C00682=1031.531,281.034,-121.463,170.893,45.172,158.687
C00683=1031.524,280.786,-121.432,170.889,45.173,158.687
C00684=1031.517,280.538,-121.401,170.885,45.173,158.687
C00685=1031.510,280.290,-121.369,170.881,45.172,158.686
C00686=1031.503,280.042,-121.338,170.877,45.173,158.686
C00687=1031.497,279.794,-121.307,170.873,45.173,158.685
C00688=1031.490,279.546,-121.275,170.870,45.173,158.685
C00689=1031.484,279.298,-121.244,170.865,45.173,158.685
C00690=1031.477,279.050,-121.213,170.862,45.173,158.684
C00691=1031.471,278.802,-121.182,170.858,45.173,158.684
C00692=1031.464,278.554,-121.151,170.855,45.174,158.684
C00693=1031.458,278.306,-121.119,170.850,45.174,158.683
C00694=1031.447,277.940,-121.074,170.845,45.174,158.683
C00695=1031.437,277.573,-121.027,170.839,45.174,158.682
C00696=1031.427,277.207,-120.983,170.833,45.175,158.682
C00697=1031.417,276.840,-120.937,170.827,45.175,158.681
C00698=1031.411,276.592,-120.905,170.824,45.175,158.681
C00699=1031.403,276.344,-120.875,170.820,45.175,158.680
C00700=1031.397,276.096,-120.844,170.817,45.175,158.680
C00701=1031.391,275.848,-120.813,170.813,45.176,158.680
C00702=1031.383,275.601,-120.782,170.809,45.176,158.679
C00703=1031.377,275.352,-120.752,170.805,45.177,158.679
C00704=1031.370,275.104,-120.720,170.802,45.177,158.679
C00705=1031.363,274.856,-120.690,170.797,45.177,158.678
C00706=1031.356,274.608,-120.659,170.794,45.177,158.678
C00707=1031.351,274.360,-120.628,170.790,45.177,158.678
C00708=1031.343,274.113,-120.597,170.786,45.177,158.677
C00709=1031.337,273.864,-120.567,170.782,45.178,158.677
C00710=1031.329,273.616,-120.536,170.779,45.178,158.677
C00711=1031.323,273.368,-120.505,170.775,45.178,158.676
C00712=1031.317,273.120,-120.475,170.772,45.179,158.676
C00713=1031.310,272.873,-120.444,170.767,45.179,158.676
C00714=1031.303,272.624,-120.413,170.764,45.179,158.675
C00715=1031.296,272.376,-120.383,170.760,45.180,158.675
C00716=1031.290,272.129,-120.352,170.757,45.180,158.675
C00717=1031.283,271.880,-120.322,170.752,45.180,158.675
C00718=1031.276,271.632,-120.291,170.749,45.180,158.674
C00719=1031.270,271.383,-120.261,170.745,45.181,158.674
C00720=1031.263,271.136,-120.230,170.742,45.181,158.674
C00721=1031.257,270.888,-120.199,170.737,45.181,158.673
C00722=1031.249,270.640,-120.169,170.734,45.181,158.673
C00723=1031.243,270.391,-120.139,170.730,45.182,158.673
C00724=1031.236,270.144,-120.108,170.727,45.182,158.672
C00725=1031.230,269.896,-120.077,170.723,45.183,158.672
C00726=1031.223,269.648,-120.047,170.719,45.183,158.672
C00727=1031.216,269.400,-120.017,170.716,45.183,158.672
C00728=1031.210,269.151,-119.987,170.712,45.184,158.671
C00729=1031.202,268.903,-119.957,170.709,45.184,158.671
C00730=1031.197,268.655,-119.926,170.704,45.185,158.671
C00731=1031.189,268.407,-119.896,170.701,45.185,158.670
C00732=1031.182,268.160,-119.865,170.697,45.186,158.670
C00733=1031.176,267.911,-119.835,170.694,45.186,158.670
C00734=1031.169,267.664,-119.805,170.691,45.186,158.670
C00735=1031.162,267.415,-119.775,170.687,45.187,158.669
C00736=1031.156,267.168,-119.744,170.683,45.187,158.669
C00737=1031.149,266.919,-119.714,170.679,45.188,158.669
C00738=1031.142,266.671,-119.684,170.676,45.188,158.668
C00739=1031.136,266.423,-119.654,170.672,45.189,158.668
C00740=1031.129,266.175,-119.624,170.669,45.189,158.668
C00741=1031.122,265.926,-119.594,170.666,45.189,158.668
C00742=1031.116,265.678,-119.564,170.661,45.190,158.667
C00743=1031.109,265.430,-119.534,170.658,45.190,158.667
C00744=1031.102,265.182,-119.504,170.654,45.191,158.667
C00745=1031.095,264.935,-119.474,170.651,45.191,158.666
C00746=1031.089,264.686,-119.443,170.647,45.192,158.666
C00747=1031.082,264.439,-119.413,170.643,45.192,158.666
C00748=1031.075,264.190,-119.384,170.640,45.192,158.666
C00749=1031.068,263.941,-119.354,170.636,45.193,158.666
C00750=1031.059,263.580,-119.311,170.631,45.194,158.665
C00751=1031.049,263.219,-119.266,170.626,45.194,158.665
C00752=1031.040,262.856,-119.222,170.620,45.195,158.664
C00753=1031.030,262.494,-119.179,170.615,45.196,158.664
C00754=1031.023,262.246,-119.149,170.612,45.196,158.664
C00755=1031.017,261.998,-119.120,170.609,45.197,158.663
C00756=1031.010,261.750,-119.089,170.605,45.197,158.663
C00757=1031.004,261.502,-119.059,170.601,45.198,158.663
C00758=1030.997,261.253,-119.030,170.598,45.198,158.663
C00759=1030.990,261.006,-119.000,170.594,45.199,158.662
C00760=1030.983,260.758,-118.970,170.591,45.199,158.662
C00761=1030.976,260.510,-118.941,170.587,45.200,158.662
C00762=1030.969,260.261,-118.911,170.584,45.201,158.662
C00763=1030.962,260.013,-118.882,170.581,45.201,158.662
C00764=1030.956,259.765,-118.852,170.577,45.202,158.661
C00765=1030.949,259.516,-118.823,170.574,45.203,158.661
C00766=1030.942,259.269,-118.793,170.570,45.203,158.661
C00767=1030.935,259.020,-118.764,170.566,45.203,158.661
C00768=1030.928,258.772,-118.735,170.563,45.204,158.660
C00769=1030.921,258.524,-118.705,170.559,45.205,158.660
C00770=1030.915,258.276,-118.676,170.556,45.206,158.660
C00771=1030.908,258.027,-118.646,170.552,45.207,158.660
C00772=1030.901,257.780,-118.617,170.549,45.207,158.660
C00773=1030.894,257.531,-118.588,170.546,45.207,158.659
C00774=1030.888,257.283,-118.558,170.542,45.208,158.659
C00775=1030.881,257.034,-118.529,170.539,45.209,158.659
C00776=1030.874,256.787,-118.499,170.535,45.210,158.659
C00777=1030.867,256.538,-118.470,170.531,45.210,158.658
C00778=1030.860,256.290,-118.441,170.528,45.211,158.658
C00779=1030.853,256.042,-118.411,170.524,45.212,158.658
C00780=1030.847,255.794,-118.382,170.521,45.212,158.658
C00781=1030.841,255.546,-118.353,170.518,45.213,158.658
C00782=1030.834,255.297,-118.324,170.514,45.214,158.658
C00783=1030.826,255.050,-118.294,170.511,45.214,158.657
C00784=1030.820,254.801,-118.265,170.508,45.215,158.657
C00785=1030.813,254.553,-118.236,170.504,45.215,158.657
C00786=1030.807,254.305,-118.207,170.501,45.216,158.657
C00787=1030.800,254.057,-118.177,170.498,45.217,158.656
C00788=1030.794,253.808,-118.148,170.494,45.218,158.656
C00789=1030.786,253.560,-118.119,170.491,45.218,158.656
C00790=1030.780,253.312,-118.090,170.488,45.219,158.656
C00791=1030.774,253.064,-118.061,170.483,45.219,158.656
C00792=1030.766,252.815,-118.031,170.480,45.220,158.655
C00793=1030.760,252.567,-118.002,170.477,45.221,158.655
C00794=1030.753,252.319,-117.973,170.473,45.222,158.655
C00795=1030.746,252.071,-117.944,170.470,45.222,158.655
C00796=1030.740,251.822,-117.915,170.467,45.223,158.655
C00797=1030.734,251.574,-117.886,170.464,45.224,158.655
C00798=1030.727,251.325,-117.856,170.460,45.225,158.654
C00799=1030.720,251.078,-117.827,170.457,45.225,158.654
C00800=1030.713,250.830,-117.798,170.454,45.226,158.654
C00801=1030.707,250.581,-117.769,170.450,45.227,158.654
C00802=1030.700,250.333,-117.740,170.447,45.227,158.653
C00803=1030.694,250.085,-117.711,170.444,45.228,158.653
C00804=1030.687,249.837,-117.682,170.441,45.228,158.653
C00805=1030.680,249.588,-117.653,170.437,45.229,158.653
C00806=1030.671,249.225,-117.610,170.433,45.230,158.653
C00807=1030.661,248.862,-117.567,170.427,45.231,158.652
C00808=1030.652,248.498,-117.525,170.422,45.232,158.652
C00809=1030.643,248.135,-117.483,170.417,45.234,158.652
C00810=1030.635,247.887,-117.454,170.414,45.234,158.652
C00811=1030.629,247.639,-117.425,170.411,45.235,158.652
C00812=1030.623,247.390,-117.396,170.408,45.236,158.651
C00813=1030.616,247.142,-117.367,170.404,45.237,158.651
C00814=1030.610,246.894,-117.338,170.401,45.237,158.651
C00815=1030.603,246.646,-117.309,170.398,45.238,158.651
C00816=1030.596,246.397,-117.280,170.395,45.239,158.651
C00817=1030.590,246.149,-117.251,170.391,45.240,158.650
C00818=1030.584,245.901,-117.222,170.388,45.240,158.650
C00819=1030.577,245.653,-117.195,170.385,45.241,158.650
C00820=1030.570,245.404,-117.165,170.382,45.242,158.650
C00821=1030.564,245.156,-117.136,170.379,45.242,158.650
C00822=1030.558,244.908,-117.107,170.375,45.243,158.650
C00823=1030.552,244.660,-117.078,170.372,45.244,158.649
C00824=1030.545,244.412,-117.050,170.369,45.245,158.649
C00825=1030.539,244.163,-117.021,170.366,45.245,158.649
C00826=1030.532,243.915,-116.993,170.363,45.246,158.649
C00827=1030.525,243.666,-116.963,170.359,45.247,158.649
C00828=1030.518,243.418,-116.936,170.356,45.248,158.648
C00829=1030.512,243.170,-116.907,170.353,45.249,158.648
C00830=1030.505,242.922,-116.878,170.350,45.250,158.648
C00831=1030.499,242.673,-116.850,170.346,45.250,158.648
C00832=1030.492,242.425,-116.821,170.343,45.251,158.648
C00833=1030.485,242.177,-116.792,170.340,45.252,158.648
C00834=1030.478,241.928,-116.764,170.337,45.252,158.648
C00835=1030.472,241.680,-116.735,170.334,45.254,158.648
C00836=1030.465,241.432,-116.707,170.330,45.255,158.647
C00837=1030.459,241.183,-116.678,170.327,45.255,158.647
C00838=1030.452,240.936,-116.650,170.324,45.256,158.647
C00839=1030.446,240.687,-116.622,170.321,45.257,158.647
C00840=1030.439,240.439,-116.593,170.318,45.258,158.647
C00841=1030.433,240.190,-116.565,170.314,45.259,158.647
C00842=1030.426,239.942,-116.536,170.311,45.260,158.647
C00843=1030.419,239.693,-116.508,170.308,45.260,158.646
C00844=1030.413,239.445,-116.479,170.305,45.262,158.646
C00845=1030.406,239.197,-116.452,170.301,45.263,158.646
C00846=1030.399,238.949,-116.423,170.298,45.263,158.646
C00847=1030.393,238.700,-116.395,170.295,45.265,158.646
C00848=1030.387,238.452,-116.367,170.292,45.265,158.646
C00849=1030.380,238.204,-116.339,170.289,45.266,158.646
C00850=1030.373,237.955,-116.311,170.285,45.268,158.646
C00851=1030.366,237.708,-116.282,170.282,45.268,158.645
C00852=1030.360,237.459,-116.254,170.279,45.269,158.645
C00853=1030.353,237.210,-116.226,170.276,45.270,158.645
C00854=1030.346,236.962,-116.198,170.273,45.271,158.645
C00855=1030.339,236.713,-116.170,170.269,45.272,158.645
C00856=1030.332,236.465,-116.142,170.267,45.273,158.645
C00857=1030.326,236.217,-116.114,170.264,45.274,158.645
C00858=1030.319,235.968,-116.085,170.261,45.275,158.645
C00859=1030.313,235.720,-116.058,170.258,45.276,158.644
C00860=1030.306,235.472,-116.030,170.254,45.277,158.644
C00861=1030.299,235.224,-116.001,170.251,45.278,158.644
C00862=1030.289,234.854,-115.960,170.247,45.279,158.644
C00863=1030.279,234.485,-115.918,170.242,45.281,158.644
C00864=1030.269,234.116,-115.877,170.237,45.283,158.644
C00865=1030.260,233.746,-115.835,170.232,45.284,158.644
C00866=1030.254,233.498,-115.807,170.229,45.285,158.644
C00867=1030.247,233.249,-115.779,170.226,45.286,158.643
C00868=1030.240,233.001,-115.752,170.223,45.286,158.643
C00869=1030.234,232.752,-115.724,170.221,45.288,158.643
C00870=1030.227,232.505,-115.695,170.218,45.288,158.643
C00871=1030.220,232.256,-115.668,170.214,45.290,158.643
C00872=1030.215,232.008,-115.640,170.211,45.291,158.643
C00873=1030.208,231.760,-115.612,170.208,45.292,158.643
C00874=1030.201,231.511,-115.584,170.205,45.293,158.643
C00875=1030.195,231.263,-115.557,170.202,45.294,158.643
C00876=1030.188,231.014,-115.529,170.199,45.295,158.642
C00877=1030.181,230.766,-115.501,170.196,45.296,158.642
C00878=1030.174,230.517,-115.473,170.192,45.297,158.642
C00879=1030.168,230.269,-115.446,170.190,45.298,158.642
C00880=1030.161,230.021,-115.418,170.187,45.299,158.642
C00881=1030.154,229.772,-115.390,170.184,45.300,158.642
C00882=1030.148,229.524,-115.362,170.181,45.301,158.642
C00883=1030.141,229.275,-115.335,170.178,45.302,158.642
C00884=1030.134,229.027,-115.307,170.175,45.303,158.642
C00885=1030.128,228.779,-115.280,170.172,45.304,158.642
C00886=1030.122,228.531,-115.252,170.168,45.305,158.641
C00887=1030.115,228.282,-115.224,170.165,45.307,158.641
C00888=1030.108,228.034,-115.196,170.162,45.307,158.641
C00889=1030.102,227.785,-115.169,170.159,45.309,158.641
C00890=1030.095,227.537,-115.141,170.157,45.310,158.641
C00891=1030.088,227.288,-115.113,170.154,45.311,158.641
C00892=1030.082,227.039,-115.086,170.151,45.312,158.641
C00893=1030.075,226.792,-115.059,170.147,45.313,158.641
C00894=1030.068,226.543,-115.032,170.144,45.314,158.641
C00895=1030.062,226.295,-115.004,170.141,45.315,158.641
C00896=1030.055,226.047,-114.976,170.139,45.317,158.641
C00897=1030.048,225.798,-114.950,170.135,45.317,158.641
C00898=1030.041,225.549,-114.922,170.133,45.319,158.641
C00899=1030.034,225.301,-114.894,170.130,45.320,158.641
C00900=1030.029,225.053,-114.868,170.127,45.321,158.641
C00901=1030.022,224.804,-114.840,170.123,45.322,158.640
C00902=1030.015,224.556,-114.813,170.120,45.324,158.640
C00903=1030.008,224.308,-114.785,170.117,45.324,158.640
C00904=1030.002,224.059,-114.758,170.114,45.326,158.640
C00905=1029.995,223.810,-114.730,170.112,45.327,158.640
C00906=1029.988,223.563,-114.704,170.109,45.328,158.640
C00907=1029.982,223.314,-114.677,170.106,45.329,158.640
C00908=1029.975,223.065,-114.649,170.103,45.330,158.640
C00909=1029.968,222.817,-114.621,170.100,45.332,158.640
C00910=1029.961,222.568,-114.595,170.096,45.333,158.640
C00911=1029.955,222.320,-114.567,170.094,45.334,158.640
C00912=1029.948,222.072,-114.540,170.091,45.335,158.640
C00913=1029.942,221.823,-114.513,170.088,45.336,158.640
C00914=1029.935,221.575,-114.486,170.085,45.337,158.640
C00915=1029.928,221.326,-114.458,170.082,45.339,158.640
C00916=1029.922,221.078,-114.431,170.079,45.340,158.640
C00917=1029.916,220.829,-114.403,170.076,45.341,158.640
C00918=1029.906,220.453,-114.362,170.072,45.342,158.639
C00919=1029.895,220.075,-114.321,170.068,45.345,158.640
C00920=1029.885,219.699,-114.280,170.063,45.346,158.639
C00921=1029.875,219.321,-114.239,170.058,45.348,158.639
C00922=1029.869,219.073,-114.212,170.056,45.350,158.639
C00923=1029.862,218.824,-114.186,170.053,45.351,158.639
C00924=1029.855,218.576,-114.158,170.050,45.352,158.639
C00925=1029.849,218.328,-114.132,170.047,45.353,158.639
C00926=1029.842,218.079,-114.104,170.044,45.354,158.639
C00927=1029.835,217.831,-114.078,170.042,45.356,158.639
C00928=1029.829,217.581,-114.051,170.039,45.357,158.639
C00929=1029.822,217.334,-114.024,170.036,45.358,158.639
C00930=1029.815,217.085,-113.997,170.032,45.360,158.639
C00931=1029.808,216.836,-113.971,170.029,45.361,158.639
C00932=1029.802,216.589,-113.943,170.026,45.362,158.639
C00933=1029.795,216.340,-113.917,170.024,45.363,158.639
C00934=1029.788,216.091,-113.890,170.021,45.364,158.639
C00935=1029.781,215.843,-113.863,170.018,45.366,158.639
C00936=1029.775,215.595,-113.837,170.015,45.367,158.639
C00937=1029.768,215.345,-113.810,170.012,45.368,158.639
C00938=1029.761,215.097,-113.782,170.010,45.370,158.639
C00939=1029.755,214.849,-113.756,170.007,45.371,158.639
C00940=1029.748,214.600,-113.729,170.004,45.372,158.639
C00941=1029.742,214.351,-113.702,170.001,45.374,158.639
C00942=1029.735,214.104,-113.676,169.999,45.375,158.639
C00943=1029.729,213.855,-113.649,169.996,45.376,158.639
C00944=1029.722,213.607,-113.623,169.993,45.377,158.639
C00945=1029.716,213.358,-113.596,169.990,45.379,158.639
C00946=1029.708,213.109,-113.568,169.987,45.380,158.639
C00947=1029.702,212.861,-113.542,169.984,45.381,158.639
C00948=1029.695,212.612,-113.515,169.981,45.383,158.638
C00949=1029.688,212.364,-113.489,169.978,45.384,158.638
C00950=1029.682,212.115,-113.462,169.975,45.385,158.638
C00951=1029.675,211.867,-113.435,169.972,45.387,158.638
C00952=1029.669,211.619,-113.408,169.970,45.388,158.638
C00953=1029.662,211.370,-113.382,169.967,45.389,158.638
C00954=1029.656,211.122,-113.355,169.964,45.391,158.638
C00955=1029.649,210.873,-113.329,169.961,45.392,158.638
C00956=1029.642,210.624,-113.303,169.958,45.393,158.638
C00957=1029.636,210.376,-113.276,169.956,45.395,158.638
C00958=1029.629,210.127,-113.250,169.953,45.396,158.638
C00959=1029.623,209.879,-113.223,169.950,45.397,158.638
C00960=1029.616,209.630,-113.197,169.947,45.399,158.638
C00961=1029.609,209.381,-113.170,169.945,45.400,158.638
C00962=1029.602,209.134,-113.143,169.942,45.401,158.638
C00963=1029.595,208.885,-113.117,169.939,45.403,158.638
C00964=1029.589,208.637,-113.091,169.936,45.404,158.638
C00965=1029.582,208.388,-113.064,169.933,45.405,158.638
C00966=1029.576,208.139,-113.038,169.931,45.407,158.638
C00967=1029.569,207.890,-113.012,169.928,45.408,158.638
C00968=1029.563,207.642,-112.986,169.925,45.409,158.638
C00969=1029.556,207.394,-112.960,169.922,45.411,158.638
C00970=1029.549,207.145,-112.933,169.920,45.413,158.638
C00971=1029.543,206.897,-112.906,169.917,45.414,158.638
C00972=1029.536,206.648,-112.880,169.914,45.415,158.638
C00973=1029.529,206.400,-112.854,169.912,45.417,158.638
C00974=1029.519,206.028,-112.815,169.907,45.419,158.638
C00975=1029.509,205.657,-112.776,169.903,45.421,158.638
C00976=1029.499,205.286,-112.737,169.899,45.423,158.638
C00977=1029.488,204.914,-112.698,169.895,45.425,158.639
C00978=1029.463,203.867,-112.593,169.531,45.322,158.579
C00979=1029.457,203.619,-112.569,169.528,45.324,158.579
C00980=1029.451,203.370,-112.543,169.524,45.326,158.579
C00981=1029.445,203.121,-112.519,169.520,45.328,158.579
C00982=1029.440,202.873,-112.494,169.516,45.331,158.579
C00983=1029.434,202.623,-112.469,169.512,45.333,158.579
C00984=1029.427,202.375,-112.444,169.509,45.335,158.579
C00985=1029.422,202.126,-112.420,169.505,45.337,158.579
C00986=1029.416,201.877,-112.395,169.502,45.340,158.579
C00987=1029.410,201.628,-112.370,169.497,45.342,158.579
C00988=1029.404,201.380,-112.346,169.493,45.344,158.579
C00989=1029.398,201.131,-112.321,169.490,45.346,158.579
C00990=1029.392,200.883,-112.297,169.486,45.348,158.580
C00991=1029.386,200.634,-112.272,169.483,45.350,158.580
C00992=1029.380,200.385,-112.247,169.479,45.352,158.580
C00993=1029.375,200.136,-112.223,169.476,45.355,158.580
C00994=1029.368,199.887,-112.199,169.471,45.358,158.580
C00995=1029.362,199.639,-112.173,169.468,45.360,158.580
C00996=1029.356,199.390,-112.150,169.464,45.362,158.580
C00997=1029.350,199.141,-112.125,169.461,45.364,158.580
C00998=1029.343,198.892,-112.101,169.457,45.367,158.580
C00999=1029.338,198.644,-112.077,169.453,45.369,158.580
C01000=1029.331,198.395,-112.052,169.449,45.372,158.581
C01001=1029.326,198.147,-112.028,169.446,45.374,158.581
C01002=1029.319,197.898,-112.004,169.442,45.376,158.581
C01003=1029.313,197.648,-111.979,169.439,45.379,158.581
C01004=1029.307,197.400,-111.955,169.434,45.381,158.581
C01005=1029.300,197.151,-111.931,169.431,45.383,158.581
C01006=1029.295,196.903,-111.907,169.427,45.386,158.581
C01007=1029.288,196.654,-111.882,169.424,45.388,158.581
C01008=1029.283,196.406,-111.858,169.420,45.390,158.581
C01009=1029.276,196.157,-111.834,169.417,45.393,158.581
C01010=1029.271,195.908,-111.810,169.413,45.395,158.582
C01011=1029.264,195.659,-111.786,169.409,45.398,158.582
C01012=1029.259,195.410,-111.762,169.405,45.400,158.582
C01013=1029.252,195.161,-111.738,169.402,45.402,158.582
C01014=1029.246,194.912,-111.713,169.398,45.405,158.582
C01015=1029.240,194.664,-111.689,169.395,45.408,158.582
C01016=1029.235,194.415,-111.665,169.392,45.410,158.582
C01017=1029.228,194.166,-111.641,169.388,45.412,158.582
C01018=1029.222,193.918,-111.617,169.384,45.414,158.582
C01019=1029.217,193.669,-111.593,169.381,45.416,158.583
C01020=1029.211,193.420,-111.569,169.378,45.419,158.583
C01021=1029.205,193.171,-111.544,169.373,45.422,158.583
C01022=1029.199,192.923,-111.521,169.370,45.424,158.583
C01023=1029.193,192.674,-111.496,169.366,45.426,158.583
C01024=1029.187,192.425,-111.472,169.363,45.429,158.583
C01025=1029.181,192.176,-111.448,169.359,45.431,158.583
C01026=1029.175,191.927,-111.425,169.356,45.433,158.583
C01027=1029.168,191.678,-111.401,169.352,45.436,158.583
C01028=1029.163,191.430,-111.377,169.349,45.439,158.584
C01029=1029.157,191.181,-111.353,169.345,45.441,158.584
C01030=1029.151,190.932,-111.328,169.342,45.443,158.584
C01031=1029.145,190.684,-111.305,169.338,45.445,158.584
C01032=1029.139,190.434,-111.280,169.335,45.448,158.584
C01033=1029.133,190.186,-111.256,169.331,45.450,158.584
C01034=1029.127,189.937,-111.233,169.328,45.453,158.584
C01035=1029.122,189.688,-111.209,169.325,45.455,158.585
C01036=1029.115,189.440,-111.185,169.321,45.458,158.585
C01037=1029.110,189.191,-111.161,169.318,45.460,158.585
C01038=1029.104,188.942,-111.137,169.314,45.462,158.585
C01039=1029.098,188.659,-111.110,169.310,45.465,158.585
C01040=1029.091,188.375,-111.083,169.305,45.468,158.585
C01041=1029.084,188.093,-111.056,169.302,45.471,158.585
C01042=1029.078,187.809,-111.029,169.298,45.474,158.585
C01043=1029.072,187.560,-111.005,169.294,45.476,158.586
C01044=1029.066,187.311,-110.981,169.291,45.478,158.586
C01045=1029.060,187.063,-110.957,169.287,45.481,158.586
C01046=1029.055,186.814,-110.933,169.284,45.483,158.586
C01047=1029.048,186.565,-110.909,169.280,45.485,158.586
C01048=1029.042,186.316,-110.886,169.277,45.488,158.586
C01049=1029.037,186.067,-110.862,169.273,45.490,158.586
C01050=1029.031,185.819,-110.838,169.271,45.492,158.586
C01051=1029.025,185.570,-110.814,169.267,45.495,158.587
C01052=1029.019,185.321,-110.791,169.264,45.498,158.587
C01053=1029.013,185.072,-110.767,169.260,45.500,158.587
C01054=1029.008,184.823,-110.744,169.257,45.502,158.587
C01055=1029.002,184.574,-110.720,169.254,45.505,158.587
C01056=1028.996,184.326,-110.695,169.250,45.507,158.587
C01057=1028.991,184.077,-110.672,169.247,45.509,158.587
C01058=1028.985,183.828,-110.649,169.243,45.512,158.588
C01059=1028.980,183.579,-110.625,169.240,45.515,158.588
C01060=1028.973,183.330,-110.601,169.236,45.517,158.588
C01061=1028.968,183.081,-110.578,169.233,45.520,158.588
C01062=1028.962,182.833,-110.554,169.229,45.522,158.588
C01063=1028.956,182.584,-110.531,169.226,45.525,158.588
C01064=1028.950,182.335,-110.507,169.223,45.527,158.588
C01065=1028.943,182.086,-110.485,169.219,45.530,158.589
C01066=1028.937,181.837,-110.462,169.216,45.533,158.589
C01067=1028.931,181.589,-110.438,169.213,45.535,158.589
C01068=1028.925,181.340,-110.415,169.209,45.538,158.589
C01069=1028.919,181.091,-110.392,169.206,45.541,158.589
C01070=1028.913,180.842,-110.369,169.202,45.543,158.589
C01071=1028.907,180.594,-110.346,169.199,45.546,158.590
C01072=1028.900,180.344,-110.322,169.196,45.548,158.590
C01073=1028.895,180.095,-110.300,169.192,45.551,158.590
C01074=1028.889,179.846,-110.277,169.189,45.554,158.590
C01075=1028.882,179.598,-110.254,169.186,45.556,158.590
C01076=1028.876,179.349,-110.230,169.182,45.559,158.591
C01077=1028.870,179.100,-110.207,169.179,45.562,158.591
C01078=1028.864,178.851,-110.184,169.175,45.564,158.591
C01079=1028.859,178.602,-110.161,169.172,45.567,158.591
C01080=1028.852,178.354,-110.139,169.169,45.570,158.591
C01081=1028.846,178.105,-110.115,169.165,45.572,158.591
C01082=1028.840,177.856,-110.092,169.162,45.575,158.592
C01083=1028.834,177.607,-110.069,169.159,45.578,158.592
C01084=1028.828,177.358,-110.046,169.155,45.580,158.592
C01085=1028.822,177.109,-110.024,169.152,45.583,158.592
C01086=1028.816,176.860,-110.001,169.150,45.586,158.593
C01087=1028.810,176.611,-109.978,169.146,45.588,158.593
C01088=1028.804,176.362,-109.955,169.143,45.591,158.593
C01089=1028.798,176.113,-109.932,169.140,45.594,158.593
C01090=1028.792,175.864,-109.909,169.136,45.596,158.593
C01091=1028.786,175.615,-109.886,169.133,45.599,158.593
C01092=1028.780,175.367,-109.863,169.130,45.602,158.594
C01093=1028.774,175.118,-109.840,169.126,45.605,158.594
C01094=1028.768,174.870,-109.817,169.123,45.607,158.594
C01095=1028.762,174.621,-109.794,169.120,45.610,158.594
C01096=1028.756,174.371,-109.771,169.116,45.613,158.594
C01097=1028.750,174.122,-109.748,169.113,45.615,158.594
C01098=1028.744,173.874,-109.726,169.109,45.618,158.595
C01099=1028.738,173.625,-109.703,169.107,45.621,158.595
C01100=1028.732,173.376,-109.680,169.104,45.623,158.595
C01101=1028.726,173.127,-109.657,169.100,45.626,158.595
C01102=1028.720,172.878,-109.635,169.097,45.629,158.596
C01103=1028.714,172.594,-109.609,169.093,45.632,158.596
C01104=1028.707,172.311,-109.582,169.090,45.635,158.596
C01105=1028.701,172.027,-109.557,169.086,45.638,158.596
C01106=1028.694,171.743,-109.531,169.082,45.641,158.596
C01107=1028.687,171.494,-109.508,169.079,45.644,158.597
C01108=1028.682,171.246,-109.485,169.076,45.646,158.597
C01109=1028.676,170.997,-109.462,169.073,45.648,158.597
C01110=1028.670,170.748,-109.439,169.070,45.651,158.597
C01111=1028.664,170.499,-109.418,169.066,45.654,158.597
C01112=1028.658,170.250,-109.395,169.063,45.657,158.597
C01113=1028.652,170.001,-109.372,169.060,45.659,158.598
C01114=1028.647,169.752,-109.349,169.056,45.662,158.598
C01115=1028.640,169.503,-109.327,169.054,45.664,158.598
C01116=1028.635,169.254,-109.304,169.051,45.667,158.598
C01117=1028.629,169.005,-109.281,169.047,45.670,158.599
C01118=1028.623,168.756,-109.259,169.044,45.673,158.599
C01119=1028.617,168.507,-109.236,169.041,45.675,158.599
C01120=1028.611,168.258,-109.213,169.038,45.678,158.599
C01121=1028.605,168.010,-109.190,169.035,45.681,158.599
C01122=1028.601,167.761,-109.168,169.031,45.683,158.599
C01123=1028.594,167.512,-109.146,169.028,45.686,158.600
C01124=1028.588,167.263,-109.123,169.025,45.689,158.600
C01125=1028.583,167.014,-109.100,169.021,45.691,158.600
C01126=1028.577,166.765,-109.079,169.019,45.694,158.600
C01127=1028.571,166.516,-109.056,169.016,45.697,158.600
C01128=1028.565,166.267,-109.033,169.013,45.700,158.601
C01129=1028.559,166.019,-109.010,169.009,45.702,158.601
C01130=1028.553,165.769,-108.988,169.007,45.705,158.601
C01131=1028.547,165.520,-108.965,169.004,45.708,158.601
C01132=1028.542,165.272,-108.943,169.000,45.710,158.601
C01133=1028.537,165.023,-108.920,168.997,45.713,158.602
C01134=1028.530,164.774,-108.898,168.994,45.715,158.602
C01135=1028.525,164.525,-108.875,168.991,45.718,158.602
C01136=1028.519,164.276,-108.853,168.988,45.721,158.602
C01137=1028.513,164.027,-108.830,168.984,45.723,158.602
C01138=1028.507,163.778,-108.807,168.982,45.726,158.603
C01139=1028.502,163.529,-108.786,168.979,45.728,158.603
C01140=1028.497,163.281,-108.763,168.975,45.731,158.603
C01141=1028.490,163.031,-108.741,168.972,45.734,158.603
C01142=1028.485,162.782,-108.718,168.970,45.737,158.604
C01143=1028.479,162.533,-108.695,168.966,45.739,158.604
C01144=1028.473,162.285,-108.674,168.963,45.742,158.604
C01145=1028.468,162.036,-108.651,168.960,45.745,158.604
C01146=1028.462,161.787,-108.629,168.958,45.748,158.604
C01147=1028.456,161.538,-108.606,168.954,45.750,158.604
C01148=1028.450,161.288,-108.584,168.951,45.753,158.605
C01149=1028.445,161.040,-108.562,168.948,45.756,158.605
C01150=1028.440,160.791,-108.539,168.945,45.758,158.605
C01151=1028.433,160.542,-108.517,168.942,45.761,158.605
C01152=1028.428,160.293,-108.494,168.938,45.764,158.605
C01153=1028.423,160.044,-108.472,168.936,45.766,158.606
C01154=1028.416,159.796,-108.450,168.933,45.769,158.606
C01155=1028.411,159.546,-108.428,168.929,45.771,158.606
C01156=1028.405,159.297,-108.405,168.927,45.774,158.606
C01157=1028.399,159.048,-108.383,168.924,45.777,158.607
C01158=1028.393,158.800,-108.362,168.921,45.780,158.607
C01159=1028.387,158.551,-108.340,168.917,45.783,158.607
C01160=1028.381,158.302,-108.317,168.915,45.786,158.607
C01161=1028.375,158.052,-108.295,168.912,45.789,158.608
C01162=1028.369,157.803,-108.274,168.909,45.791,158.608
C01163=1028.364,157.555,-108.253,168.905,45.794,158.608
C01164=1028.358,157.306,-108.230,168.903,45.796,158.608
C01165=1028.352,157.057,-108.208,168.900,45.799,158.608
C01166=1028.346,156.807,-108.186,168.896,45.802,158.609
C01167=1028.339,156.524,-108.161,168.893,45.806,158.609
C01168=1028.333,156.240,-108.137,168.890,45.809,158.609
C01169=1028.326,155.955,-108.111,168.886,45.812,158.609
C01170=1028.319,155.671,-108.086,168.883,45.816,158.610
C01171=1028.313,155.422,-108.064,168.879,45.818,158.610
C01172=1028.307,155.173,-108.043,168.877,45.821,158.610
C01173=1028.301,154.925,-108.022,168.874,45.824,158.610
C01174=1028.296,154.675,-107.999,168.871,45.827,158.611
C01175=1028.290,154.426,-107.977,168.867,45.829,158.611
C01176=1028.283,154.177,-107.955,168.865,45.832,158.611
C01177=1028.278,153.929,-107.934,168.862,45.835,158.611
C01178=1028.272,153.679,-107.912,168.858,45.838,158.611
C01179=1028.266,153.430,-107.890,168.856,45.840,158.612
C01180=1028.261,153.181,-107.869,168.853,45.843,158.612
C01181=1028.255,152.932,-107.847,168.850,45.846,158.612
C01182=1028.248,152.683,-107.826,168.846,45.849,158.612
C01183=1028.243,152.435,-107.804,168.844,45.852,158.613
C01184=1028.237,152.185,-107.783,168.841,45.855,158.613
C01185=1028.230,151.936,-107.761,168.838,45.858,158.613
C01186=1028.225,151.687,-107.739,168.835,45.861,158.613
C01187=1028.219,151.438,-107.718,168.832,45.863,158.614
C01188=1028.213,151.189,-107.696,168.829,45.866,158.614
C01189=1028.207,150.940,-107.674,168.827,45.870,158.614
C01190=1028.202,150.691,-107.653,168.824,45.873,158.615
C01191=1028.195,150.442,-107.631,168.820,45.876,158.615
C01192=1028.190,150.194,-107.610,168.817,45.879,158.615
C01193=1028.184,149.944,-107.588,168.815,45.881,158.615
C01194=1028.178,149.695,-107.567,168.812,45.884,158.616
C01195=1028.172,149.447,-107.546,168.808,45.887,158.616
C01196=1028.167,149.197,-107.523,168.806,45.890,158.616
C01197=1028.160,148.948,-107.502,168.803,45.893,158.616
C01198=1028.155,148.699,-107.480,168.800,45.896,158.616
C01199=1028.149,148.450,-107.459,168.797,45.898,158.617
C01200=1028.143,148.202,-107.438,168.794,45.901,158.617
C01201=1028.137,147.952,-107.416,168.791,45.904,158.617
C01202=1028.131,147.703,-107.394,168.789,45.907,158.617
C01203=1028.126,147.454,-107.374,168.785,45.910,158.618
C01204=1028.119,147.205,-107.352,168.782,45.913,158.618
C01205=1028.114,146.956,-107.331,168.780,45.916,158.618
C01206=1028.108,146.707,-107.309,168.777,45.918,158.618
C01207=1028.101,146.458,-107.288,168.773,45.921,158.619
C01208=1028.096,146.210,-107.266,168.771,45.924,158.619
C01209=1028.090,145.960,-107.245,168.768,45.927,158.619
C01210=1028.084,145.711,-107.225,168.765,45.930,158.619
C01211=1028.078,145.462,-107.203,168.763,45.933,158.620
C01212=1028.071,145.213,-107.181,168.759,45.936,158.620
C01213=1028.066,144.964,-107.161,168.756,45.939,158.620
C01214=1028.060,144.715,-107.139,168.754,45.942,158.621
C01215=1028.054,144.466,-107.118,168.751,45.945,158.621
C01216=1028.048,144.217,-107.098,168.747,45.948,158.621
C01217=1028.042,143.968,-107.076,168.745,45.951,158.621
C01218=1028.036,143.719,-107.055,168.742,45.953,158.622
C01219=1028.030,143.469,-107.034,168.739,45.957,158.622
C01220=1028.025,143.221,-107.013,168.737,45.960,158.622
C01221=1028.019,142.971,-106.991,168.733,45.963,158.622
C01222=1028.013,142.723,-106.971,168.730,45.966,158.623
C01223=1028.006,142.473,-106.949,168.728,45.968,158.623
C01224=1028.001,142.225,-106.928,168.725,45.971,158.623
C01225=1027.995,141.975,-106.907,168.722,45.974,158.623
C01226=1027.989,141.727,-106.886,168.719,45.977,158.624
C01227=1027.983,141.478,-106.865,168.716,45.981,158.624
C01228=1027.977,141.229,-106.844,168.714,45.983,158.624
C01229=1027.971,140.979,-106.823,168.711,45.986,158.625
C01230=1027.966,140.730,-106.802,168.707,45.989,158.625
C01231=1027.959,140.446,-106.778,168.704,45.992,158.625
C01232=1027.952,140.161,-106.754,168.701,45.996,158.625
C01233=1027.945,139.877,-106.730,168.698,45.999,158.626
C01234=1027.939,139.593,-106.706,168.695,46.002,158.626
C01235=1027.933,139.344,-106.685,168.692,46.005,158.626
C01236=1027.927,139.095,-106.664,168.689,46.008,158.626
C01237=1027.921,138.845,-106.643,168.686,46.011,158.627
C01238=1027.916,138.597,-106.621,168.684,46.014,158.627
C01239=1027.909,138.347,-106.601,168.681,46.017,158.627
C01240=1027.904,138.098,-106.580,168.678,46.020,158.628
C01241=1027.898,137.850,-106.559,168.675,46.023,158.628
C01242=1027.892,137.600,-106.539,168.672,46.026,158.628
C01243=1027.886,137.352,-106.518,168.669,46.029,158.628
C01244=1027.880,137.102,-106.497,168.667,46.032,158.629
C01245=1027.874,136.854,-106.476,168.664,46.035,158.629
C01246=1027.868,136.604,-106.455,168.661,46.038,158.629
C01247=1027.862,136.355,-106.435,168.658,46.041,158.629
C01248=1027.856,136.106,-106.413,168.655,46.044,158.630
C01249=1027.851,135.857,-106.393,168.653,46.047,158.630
C01250=1027.845,135.608,-106.373,168.650,46.050,158.630
C01251=1027.838,135.359,-106.351,168.647,46.053,158.631
C01252=1027.832,135.110,-106.331,168.644,46.056,158.631
C01253=1027.827,134.860,-106.310,168.641,46.059,158.631
C01254=1027.820,134.612,-106.290,168.639,46.062,158.631
C01255=1027.815,134.363,-106.269,168.636,46.065,158.632
C01256=1027.809,134.113,-106.248,168.633,46.068,158.632
C01257=1027.803,133.865,-106.228,168.630,46.071,158.632
C01258=1027.797,133.615,-106.207,168.627,46.074,158.633
C01259=1027.791,133.366,-106.187,168.625,46.077,158.633
C01260=1027.785,133.117,-106.165,168.622,46.080,158.633
C01261=1027.779,132.868,-106.145,168.620,46.083,158.633
C01262=1027.774,132.619,-106.125,168.617,46.086,158.634
C01263=1027.768,132.370,-106.105,168.613,46.089,158.634
C01264=1027.761,132.121,-106.083,168.611,46.092,158.634
C01265=1027.755,131.872,-106.063,168.608,46.095,158.634
C01266=1027.750,131.622,-106.042,168.606,46.098,158.635
C01267=1027.744,131.373,-106.022,168.603,46.101,158.635
C01268=1027.738,131.125,-106.001,168.600,46.104,158.635
C01269=1027.732,130.875,-105.980,168.597,46.107,158.636
C01270=1027.726,130.626,-105.960,168.595,46.110,158.636
C01271=1027.721,130.377,-105.939,168.592,46.113,158.636
C01272=1027.714,130.128,-105.919,168.589,46.116,158.636
C01273=1027.708,129.879,-105.899,168.586,46.119,158.637
C01274=1027.702,129.630,-105.879,168.583,46.122,158.637
C01275=1027.696,129.380,-105.858,168.580,46.126,158.637
C01276=1027.690,129.131,-105.838,168.578,46.128,158.638
C01277=1027.684,128.882,-105.818,168.575,46.132,158.638
C01278=1027.678,128.633,-105.798,168.573,46.135,158.638
C01279=1027.672,128.384,-105.778,168.570,46.138,158.638
C01280=1027.667,128.135,-105.758,168.567,46.141,158.639
C01281=1027.660,127.885,-105.737,168.564,46.144,158.639
C01282=1027.654,127.637,-105.717,168.561,46.147,158.639
C01283=1027.648,127.388,-105.697,168.559,46.150,158.640
C01284=1027.642,127.138,-105.676,168.556,46.153,158.640
C01285=1027.636,126.889,-105.656,168.553,46.156,158.640
C01286=1027.630,126.640,-105.636,168.551,46.160,158.641
C01287=1027.624,126.391,-105.616,168.547,46.163,158.641
C01288=1027.618,126.142,-105.596,168.545,46.165,158.641
C01289=1027.612,125.893,-105.576,168.542,46.169,158.642
C01290=1027.606,125.643,-105.555,168.540,46.172,158.642
C01291=1027.600,125.395,-105.535,168.537,46.175,158.642
C01292=1027.594,125.146,-105.515,168.534,46.178,158.642
C01293=1027.588,124.897,-105.495,168.532,46.181,158.643
C01294=1027.582,124.647,-105.474,168.528,46.184,158.643
C01295=1027.575,124.363,-105.452,168.525,46.188,158.643
C01296=1027.568,124.078,-105.429,168.522,46.191,158.644
C01297=1027.561,123.794,-105.406,168.519,46.195,158.644
C01298=1027.554,123.509,-105.383,168.516,46.199,158.644
C01299=1027.549,123.260,-105.363,168.513,46.202,158.645
C01300=1027.543,123.011,-105.343,168.511,46.204,158.645
C01301=1027.537,122.762,-105.323,168.508,46.208,158.645
C01302=1027.531,122.513,-105.303,168.506,46.211,158.646
C01303=1027.525,122.264,-105.283,168.502,46.214,158.646
C01304=1027.519,122.015,-105.263,168.501,46.217,158.646
C01305=1027.513,121.766,-105.243,168.497,46.220,158.646
C01306=1027.507,121.516,-105.223,168.495,46.223,158.647
C01307=1027.501,121.267,-105.203,168.492,46.226,158.647
C01308=1027.495,121.018,-105.183,168.490,46.229,158.647
C01309=1027.490,120.769,-105.162,168.487,46.232,158.648
C01310=1027.484,120.520,-105.143,168.484,46.235,158.648
C01311=1027.477,120.270,-105.123,168.481,46.239,158.648
C01312=1027.471,120.021,-105.103,168.479,46.241,158.648
C01313=1027.465,119.772,-105.083,168.476,46.244,158.649
C01314=1027.459,119.523,-105.063,168.473,46.248,158.649
C01315=1027.454,119.274,-105.042,168.471,46.251,158.649
C01316=1027.449,119.025,-105.023,168.467,46.254,158.650
C01317=1027.443,118.776,-105.003,168.465,46.256,158.650
C01318=1027.436,118.527,-104.983,168.462,46.260,158.650
C01319=1027.430,118.278,-104.963,168.460,46.263,158.650
C01320=1027.424,118.028,-104.944,168.457,46.266,158.651
C01321=1027.419,117.779,-104.923,168.455,46.268,158.651
C01322=1027.413,117.530,-104.903,168.453,46.272,158.651
C01323=1027.407,117.281,-104.884,168.449,46.275,158.652
C01324=1027.401,117.032,-104.864,168.447,46.278,158.652
C01325=1027.395,116.783,-104.844,168.444,46.281,158.652
C01326=1027.389,116.533,-104.824,168.442,46.284,158.652
C01327=1027.384,116.284,-104.804,168.439,46.287,158.653
C01328=1027.378,116.035,-104.784,168.437,46.290,158.653
C01329=1027.372,115.786,-104.765,168.434,46.293,158.653
C01330=1027.366,115.537,-104.745,168.431,46.296,158.654
C01331=1027.360,115.288,-104.725,168.428,46.299,158.654
C01332=1027.354,115.039,-104.706,168.426,46.302,158.654
C01333=1027.349,114.790,-104.685,168.423,46.305,158.654
C01334=1027.343,114.541,-104.665,168.421,46.308,158.655
C01335=1027.338,114.291,-104.646,168.417,46.311,158.655
C01336=1027.332,114.043,-104.626,168.415,46.314,158.655
C01337=1027.325,113.792,-104.606,168.413,46.317,158.656
C01338=1027.319,113.544,-104.586,168.410,46.320,158.656
C01339=1027.314,113.295,-104.566,168.408,46.323,158.656
C01340=1027.308,113.045,-104.546,168.405,46.326,158.656
C01341=1027.302,112.796,-104.527,168.402,46.329,158.657
C01342=1027.297,112.547,-104.507,168.399,46.332,158.657
C01343=1027.291,112.298,-104.487,168.397,46.335,158.657
C01344=1027.285,112.049,-104.468,168.394,46.339,158.658
C01345=1027.278,111.800,-104.449,168.392,46.342,158.658
C01346=1027.273,111.551,-104.429,168.389,46.345,158.658
C01347=1027.267,111.301,-104.410,168.387,46.348,158.659
C01348=1027.261,111.052,-104.390,168.384,46.351,158.659
C01349=1027.255,110.803,-104.371,168.381,46.354,158.659
C01350=1027.249,110.554,-104.351,168.378,46.357,158.659
C01351=1027.243,110.304,-104.331,168.376,46.360,158.660
C01352=1027.237,110.055,-104.312,168.373,46.364,158.660
C01353=1027.230,109.806,-104.293,168.371,46.367,158.660
C01354=1027.225,109.557,-104.274,168.368,46.370,158.661
C01355=1027.219,109.307,-104.254,168.366,46.373,158.661
C01356=1027.212,109.059,-104.235,168.363,46.376,158.661
C01357=1027.207,108.809,-104.216,168.361,46.379,158.662
C01358=1027.201,108.560,-104.197,168.357,46.382,158.662
C01359=1027.194,108.276,-104.174,168.354,46.386,158.662
C01360=1027.187,107.991,-104.152,168.351,46.390,158.663
C01361=1027.181,107.706,-104.130,168.348,46.393,158.663
C01362=1027.174,107.421,-104.108,168.346,46.397,158.663
C01363=1027.167,107.173,-104.089,168.343,46.400,158.664
C01364=1027.161,106.923,-104.070,168.340,46.404,158.664
C01365=1027.156,106.674,-104.050,168.338,46.406,158.664
C01366=1027.149,106.425,-104.032,168.335,46.410,158.665
C01367=1027.143,106.176,-104.012,168.333,46.413,158.665
C01368=1027.138,105.927,-103.993,168.330,46.416,158.665
C01369=1027.131,105.677,-103.974,168.328,46.419,158.666
C01370=1027.126,105.428,-103.955,168.325,46.422,158.666
C01371=1027.120,105.179,-103.935,168.323,46.426,158.666
C01372=1027.114,104.930,-103.915,168.319,46.429,158.666
C01373=1027.107,104.681,-103.897,168.317,46.431,158.667
C01374=1027.102,104.431,-103.878,168.314,46.435,158.667
C01375=1027.096,104.182,-103.858,168.312,46.438,158.667
C01376=1027.090,103.933,-103.840,168.309,46.441,158.668
C01377=1027.084,103.684,-103.820,168.307,46.444,158.668
C01378=1027.078,103.434,-103.800,168.305,46.447,158.668
C01379=1027.072,103.185,-103.782,168.302,46.451,158.669
C01380=1027.066,102.936,-103.763,168.299,46.453,158.669
C01381=1027.060,102.686,-103.743,168.296,46.456,158.669
C01382=1027.054,102.438,-103.725,168.294,46.460,158.669
C01383=1027.049,102.189,-103.706,168.291,46.463,158.670
C01384=1027.043,101.940,-103.686,168.289,46.466,158.670
C01385=1027.036,101.691,-103.667,168.286,46.469,158.670
C01386=1027.031,101.441,-103.648,168.284,46.472,158.671
C01387=1027.025,101.192,-103.629,168.282,46.475,158.671
C01388=1027.018,100.943,-103.610,168.278,46.478,158.671
C01389=1027.013,100.693,-103.591,168.276,46.481,158.671
C01390=1027.007,100.444,-103.572,168.273,46.485,158.672
C01391=1027.001,100.195,-103.553,168.271,46.488,158.672
C01392=1026.995,99.945,-103.534,168.268,46.491,158.672
C01393=1026.990,99.696,-103.515,168.266,46.494,158.673
C01394=1026.983,99.447,-103.496,168.263,46.497,158.673
C01395=1026.978,99.198,-103.477,168.261,46.500,158.673
C01396=1026.971,98.949,-103.458,168.258,46.503,158.674
C01397=1026.965,98.700,-103.440,168.256,46.507,158.674
C01398=1026.959,98.450,-103.420,168.252,46.510,158.674
C01399=1026.953,98.201,-103.402,168.250,46.513,158.675
C01400=1026.947,97.952,-103.382,168.247,46.516,158.675
C01401=1026.941,97.703,-103.364,168.245,46.520,158.675
C01402=1026.934,97.453,-103.345,168.243,46.523,158.676
C01403=1026.929,97.205,-103.326,168.240,46.526,158.676
C01404=1026.923,96.955,-103.308,168.238,46.529,158.676
C01405=1026.917,96.706,-103.289,168.235,46.533,158.677
C01406=1026.911,96.456,-103.270,168.233,46.535,158.677
C01407=1026.904,96.207,-103.252,168.229,46.538,158.677
C01408=1026.899,95.958,-103.233,168.228,46.542,158.677
C01409=1026.892,95.709,-103.214,168.224,46.545,158.678
C01410=1026.887,95.460,-103.195,168.222,46.548,158.678
C01411=1026.881,95.210,-103.177,168.219,46.551,158.678
C01412=1026.875,94.961,-103.158,168.217,46.555,158.679
C01413=1026.869,94.712,-103.139,168.214,46.558,158.679
C01414=1026.863,94.463,-103.121,168.212,46.561,158.679
C01415=1026.857,94.213,-103.101,168.209,46.564,158.680
C01416=1026.851,93.965,-103.083,168.207,46.567,158.680
C01417=1026.845,93.715,-103.065,168.205,46.570,158.680
C01418=1026.839,93.466,-103.046,168.201,46.573,158.680
C01419=1026.833,93.216,-103.027,168.200,46.577,158.681
C01420=1026.826,92.967,-103.009,168.196,46.580,158.681
C01421=1026.821,92.719,-102.990,168.194,46.583,158.682
C01422=1026.815,92.469,-102.972,168.191,46.586,158.682
C01423=1026.808,92.184,-102.950,168.188,46.590,158.682
C01424=1026.801,91.900,-102.929,168.186,46.594,158.683
C01425=1026.795,91.615,-102.908,168.183,46.597,158.683
C01426=1026.788,91.330,-102.887,168.180,46.601,158.683
C01427=1026.782,91.081,-102.867,168.177,46.604,158.683
C01428=1026.776,90.832,-102.849,168.175,46.607,158.684
C01429=1026.770,90.583,-102.831,168.172,46.610,158.684
C01430=1026.765,90.333,-102.812,168.170,46.613,158.684
C01431=1026.758,90.084,-102.793,168.168,46.617,158.685
C01432=1026.753,89.835,-102.776,168.165,46.620,158.685
C01433=1026.747,89.586,-102.756,168.162,46.622,158.685
C01434=1026.741,89.337,-102.738,168.160,46.626,158.686
C01435=1026.734,89.087,-102.720,168.157,46.629,158.686
C01436=1026.728,88.838,-102.701,168.154,46.633,158.686
C01437=1026.722,88.589,-102.684,168.152,46.635,158.687
C01438=1026.716,88.340,-102.665,168.149,46.639,158.687
C01439=1026.710,88.090,-102.647,168.147,46.642,158.687
C01440=1026.704,87.840,-102.628,168.144,46.646,158.688
C01441=1026.699,87.591,-102.610,168.142,46.649,158.688
C01442=1026.692,87.342,-102.592,168.139,46.652,158.688
C01443=1026.686,87.093,-102.573,168.137,46.655,158.689
C01444=1026.680,86.843,-102.555,168.135,46.658,158.689
C01445=1026.674,86.595,-102.537,168.132,46.662,158.689
C01446=1026.668,86.345,-102.519,168.130,46.665,158.689
C01447=1026.661,86.096,-102.500,168.127,46.668,158.690
C01448=1026.655,85.846,-102.482,168.124,46.671,158.690
C01449=1026.649,85.598,-102.464,168.122,46.675,158.690
C01450=1026.643,85.348,-102.446,168.119,46.678,158.691
C01451=1026.637,85.098,-102.428,168.116,46.681,158.691
C01452=1026.631,84.850,-102.410,168.114,46.684,158.691
C01453=1026.625,84.600,-102.392,168.111,46.688,158.692
C01454=1026.620,84.351,-102.373,168.109,46.691,158.692
C01455=1026.614,84.102,-102.355,168.107,46.694,158.692
C01456=1026.608,83.853,-102.336,168.104,46.697,158.693
C01457=1026.601,83.603,-102.318,168.102,46.701,158.693
C01458=1026.596,83.354,-102.300,168.099,46.704,158.693
C01459=1026.590,83.105,-102.282,168.097,46.706,158.693
C01460=1026.583,82.855,-102.264,168.094,46.710,158.694
C01461=1026.578,82.607,-102.246,168.091,46.713,158.694
C01462=1026.571,82.357,-102.228,168.088,46.717,158.694
C01463=1026.565,82.108,-102.209,168.086,46.719,158.695
C01464=1026.560,81.859,-102.192,168.084,46.723,158.695
C01465=1026.553,81.609,-102.174,168.081,46.726,158.695
C01466=1026.547,81.360,-102.155,168.079,46.729,158.696
C01467=1026.541,81.111,-102.138,168.076,46.732,158.696
C01468=1026.535,80.861,-102.120,168.074,46.736,158.696
C01469=1026.529,80.612,-102.101,168.071,46.739,158.697
C01470=1026.523,80.363,-102.084,168.069,46.742,158.697
C01471=1026.518,80.113,-102.064,168.067,46.745,158.697
C01472=1026.512,79.864,-102.047,168.064,46.748,158.697
C01473=1026.506,79.615,-102.029,168.062,46.752,158.698
C01474=1026.500,79.366,-102.010,168.058,46.755,158.698
C01475=1026.494,79.116,-101.993,168.056,46.757,158.698
C01476=1026.488,78.867,-101.975,168.054,46.761,158.699
C01477=1026.482,78.618,-101.957,168.051,46.764,158.699
C01478=1026.476,78.369,-101.938,168.049,46.767,158.699
C01479=1026.470,78.119,-101.920,168.046,46.770,158.700
C01480=1026.464,77.870,-101.903,168.044,46.773,158.700
C01481=1026.458,77.620,-101.885,168.042,46.777,158.700
C01482=1026.452,77.372,-101.867,168.039,46.780,158.701
C01483=1026.446,77.122,-101.849,168.037,46.783,158.701
C01484=1026.441,76.873,-101.831,168.033,46.786,158.701
C01485=1026.434,76.623,-101.814,168.032,46.790,158.702
C01486=1026.428,76.374,-101.796,168.028,46.793,158.702
C01487=1026.421,76.089,-101.776,168.025,46.796,158.702
C01488=1026.415,75.805,-101.755,168.022,46.800,158.702
C01489=1026.408,75.520,-101.735,168.021,46.804,158.703
C01490=1026.401,75.235,-101.714,168.018,46.807,158.703
C01491=1026.394,74.986,-101.697,168.015,46.811,158.704
C01492=1026.388,74.737,-101.679,168.012,46.814,158.704
C01493=1026.382,74.488,-101.661,168.010,46.818,158.704
C01494=1026.376,74.238,-101.643,168.007,46.820,158.704
C01495=1026.370,73.989,-101.626,168.004,46.824,158.705
C01496=1026.364,73.740,-101.608,168.002,46.827,158.705
C01497=1026.358,73.490,-101.591,167.999,46.831,158.705
C01498=1026.352,73.241,-101.573,167.997,46.833,158.706
C01499=1026.346,72.992,-101.556,167.995,46.837,158.706
C01500=1026.340,72.742,-101.538,167.992,46.840,158.706
C01501=1026.334,72.493,-101.520,167.990,46.843,158.707
C01502=1026.328,72.243,-101.502,167.987,46.846,158.707
C01503=1026.323,71.994,-101.485,167.985,46.850,158.707
C01504=1026.316,71.745,-101.468,167.982,46.853,158.708
C01505=1026.310,71.495,-101.450,167.980,46.856,158.708
C01506=1026.304,71.246,-101.432,167.978,46.859,158.708
C01507=1026.298,70.996,-101.414,167.975,46.863,158.709
C01508=1026.292,70.748,-101.397,167.972,46.866,158.709
C01509=1026.286,70.498,-101.379,167.970,46.869,158.709
C01510=1026.280,70.249,-101.362,167.967,46.872,158.710
C01511=1026.274,70.000,-101.345,167.964,46.876,158.710
C01512=1026.268,69.751,-101.327,167.962,46.879,158.710
C01513=1026.262,69.501,-101.309,167.959,46.882,158.710
C01514=1026.256,69.252,-101.291,167.957,46.885,158.711
C01515=1026.250,69.003,-101.274,167.955,46.888,158.711
C01516=1026.244,68.753,-101.256,167.952,46.892,158.711
C01517=1026.238,68.504,-101.239,167.950,46.895,158.712
C01518=1026.231,68.255,-101.221,167.947,46.898,158.712
C01519=1026.226,68.006,-101.204,167.945,46.901,158.712
C01520=1026.219,67.756,-101.187,167.942,46.905,158.713
C01521=1026.214,67.507,-101.170,167.940,46.908,158.713
C01522=1026.208,67.257,-101.152,167.938,46.911,158.713
C01523=1026.201,67.008,-101.135,167.935,46.915,158.714
C01524=1026.195,66.758,-101.117,167.932,46.918,158.714
C01525=1026.189,66.510,-101.100,167.930,46.921,158.714
C01526=1026.184,66.260,-101.083,167.927,46.924,158.715
C01527=1026.177,66.011,-101.066,167.924,46.928,158.715
C01528=1026.171,65.762,-101.048,167.922,46.931,158.715
C01529=1026.165,65.512,-101.031,167.919,46.934,158.715
C01530=1026.159,65.263,-101.013,167.917,46.937,158.716
C01531=1026.153,65.013,-100.996,167.914,46.941,158.716
C01532=1026.147,64.764,-100.979,167.912,46.944,158.716
C01533=1026.142,64.515,-100.961,167.910,46.947,158.717
C01534=1026.135,64.266,-100.944,167.907,46.950,158.717
C01535=1026.129,64.016,-100.927,167.905,46.954,158.717
C01536=1026.123,63.766,-100.910,167.902,46.957,158.718
C01537=1026.117,63.517,-100.892,167.900,46.960,158.718
C01538=1026.111,63.267,-100.876,167.897,46.963,158.718
C01539=1026.104,63.019,-100.859,167.895,46.967,158.719
C01540=1026.099,62.770,-100.841,167.892,46.970,158.719
C01541=1026.092,62.520,-100.825,167.890,46.973,158.719
C01542=1026.086,62.271,-100.808,167.887,46.977,158.720
C01543=1026.079,62.021,-100.791,167.885,46.980,158.720
C01544=1026.074,61.772,-100.773,167.882,46.984,158.720
C01545=1026.067,61.522,-100.756,167.880,46.987,158.721
C01546=1026.061,61.273,-100.740,167.877,46.990,158.721
C01547=1026.055,61.024,-100.723,167.875,46.994,158.721
C01548=1026.049,60.774,-100.706,167.871,46.997,158.721
C01549=1026.043,60.525,-100.689,167.870,47.000,158.722
C01550=1026.037,60.276,-100.672,167.867,47.004,158.722
C01551=1026.029,59.991,-100.652,167.864,47.008,158.723
C01552=1026.022,59.706,-100.633,167.861,47.012,158.723
C01553=1026.015,59.421,-100.614,167.858,47.015,158.723
C01554=1026.008,59.136,-100.595,167.855,47.019,158.724
C01555=1026.002,58.887,-100.578,167.853,47.023,158.724
C01556=1025.996,58.638,-100.561,167.850,47.026,158.724
C01557=1025.990,58.388,-100.544,167.848,47.029,158.725
C01558=1025.984,58.139,-100.527,167.845,47.033,158.725
C01559=1025.978,57.890,-100.510,167.843,47.036,158.725
C01560=1025.971,57.640,-100.494,167.840,47.039,158.726
C01561=1025.965,57.391,-100.477,167.838,47.042,158.726
C01562=1025.960,57.141,-100.460,167.835,47.046,158.726
C01563=1025.953,56.892,-100.443,167.833,47.049,158.726
C01564=1025.947,56.643,-100.426,167.830,47.053,158.727
C01565=1025.941,56.394,-100.409,167.828,47.056,158.727
C01566=1025.934,56.144,-100.393,167.825,47.059,158.727
C01567=1025.929,55.894,-100.376,167.823,47.063,158.728
C01568=1025.923,55.646,-100.359,167.819,47.066,158.728
C01569=1025.916,55.395,-100.342,167.818,47.069,158.728
C01570=1025.910,55.147,-100.325,167.814,47.072,158.729
C01571=1025.905,54.897,-100.308,167.812,47.076,158.729
C01572=1025.898,54.648,-100.291,167.810,47.079,158.729
C01573=1025.892,54.398,-100.275,167.807,47.082,158.730
C01574=1025.886,54.149,-100.259,167.805,47.085,158.730
C01575=1025.880,53.900,-100.242,167.802,47.089,158.730
C01576=1025.874,53.650,-100.224,167.800,47.092,158.730
C01577=1025.868,53.400,-100.208,167.797,47.095,158.731
C01578=1025.861,53.152,-100.191,167.795,47.098,158.731
C01579=1025.856,52.902,-100.175,167.792,47.102,158.731
C01580=1025.849,52.652,-100.158,167.790,47.105,158.732
C01581=1025.843,52.403,-100.141,167.787,47.109,158.732
C01582=1025.838,52.154,-100.124,167.785,47.111,158.732
C01583=1025.832,51.905,-100.108,167.782,47.115,158.733
C01584=1025.825,51.656,-100.091,167.780,47.118,158.733
C01585=1025.819,51.406,-100.075,167.778,47.122,158.733
C01586=1025.813,51.157,-100.058,167.775,47.125,158.733
C01587=1025.807,50.907,-100.041,167.773,47.128,158.734
C01588=1025.801,50.658,-100.025,167.769,47.131,158.734
C01589=1025.795,50.409,-100.008,167.768,47.135,158.735
C01590=1025.789,50.159,-99.991,167.764,47.138,158.735
C01591=1025.783,49.910,-99.975,167.763,47.141,158.735
C01592=1025.777,49.660,-99.958,167.759,47.144,158.735
C01593=1025.771,49.411,-99.942,167.757,47.148,158.736
C01594=1025.765,49.162,-99.925,167.755,47.151,158.736
C01595=1025.759,48.912,-99.908,167.752,47.154,158.736
C01596=1025.753,48.663,-99.892,167.750,47.157,158.737
C01597=1025.747,48.413,-99.875,167.747,47.160,158.737
C01598=1025.741,48.164,-99.858,167.745,47.164,158.737
C01599=1025.735,47.915,-99.842,167.742,47.167,158.737
C01600=1025.729,47.666,-99.825,167.740,47.170,158.738
C01601=1025.723,47.416,-99.809,167.737,47.173,158.738
C01602=1025.717,47.166,-99.792,167.735,47.176,158.738
C01603=1025.711,46.917,-99.775,167.733,47.180,158.739
C01604=1025.705,46.668,-99.759,167.729,47.183,158.739
C01605=1025.699,46.419,-99.742,167.728,47.186,158.739
C01606=1025.693,46.169,-99.726,167.724,47.190,158.739
C01607=1025.687,45.920,-99.710,167.722,47.192,158.740
C01608=1025.681,45.671,-99.693,167.719,47.196,158.740
C01609=1025.675,45.421,-99.676,167.717,47.199,158.740
C01610=1025.669,45.171,-99.659,167.715,47.202,158.741
C01611=1025.663,44.922,-99.643,167.712,47.206,158.741
C01612=1025.658,44.673,-99.627,167.710,47.208,158.741
C01613=1025.652,44.423,-99.611,167.707,47.212,158.741
C01614=1025.646,44.174,-99.594,167.705,47.215,158.742
C01615=1025.639,43.889,-99.575,167.702,47.219,158.742
C01616=1025.632,43.604,-99.556,167.699,47.222,158.742
C01617=1025.625,43.318,-99.538,167.696,47.226,158.743
C01618=1025.618,43.034,-99.519,167.693,47.229,158.743
C01619=1025.613,42.784,-99.502,167.691,47.233,158.743
C01620=1025.607,42.535,-99.485,167.688,47.236,158.744
C01621=1025.600,42.286,-99.470,167.686,47.239,158.744
C01622=1025.594,42.036,-99.454,167.683,47.243,158.744
C01623=1025.588,41.787,-99.437,167.681,47.246,158.745
C01624=1025.583,41.537,-99.421,167.678,47.249,158.745
C01625=1025.577,41.288,-99.405,167.676,47.253,158.745
C01626=1025.571,41.039,-99.389,167.673,47.256,158.745
C01627=1025.564,40.788,-99.373,167.670,47.259,158.746
C01628=1025.558,40.539,-99.356,167.668,47.262,158.746
C01629=1025.552,40.289,-99.340,167.665,47.265,158.746
C01630=1025.546,40.040,-99.324,167.663,47.269,158.747
C01631=1025.540,39.791,-99.308,167.660,47.272,158.747
C01632=1025.534,39.542,-99.292,167.658,47.275,158.747
C01633=1025.528,39.292,-99.276,167.655,47.278,158.747
C01634=1025.522,39.043,-99.259,167.653,47.282,158.748
C01635=1025.516,38.794,-99.243,167.650,47.285,158.748
C01636=1025.510,38.544,-99.227,167.648,47.289,158.748
C01637=1025.504,38.295,-99.211,167.645,47.292,158.749
C01638=1025.498,38.045,-99.196,167.643,47.294,158.749
C01639=1025.492,37.796,-99.179,167.640,47.298,158.749
C01640=1025.486,37.547,-99.163,167.638,47.301,158.749
C01641=1025.480,37.297,-99.147,167.635,47.305,158.750
C01642=1025.474,37.048,-99.131,167.633,47.308,158.750
C01643=1025.468,36.799,-99.114,167.630,47.311,158.750
C01644=1025.462,36.549,-99.099,167.628,47.314,158.751
C01645=1025.456,36.300,-99.083,167.625,47.318,158.751
C01646=1025.450,36.050,-99.067,167.622,47.321,158.751
C01647=1025.443,35.801,-99.052,167.620,47.325,158.751
C01648=1025.437,35.551,-99.036,167.617,47.328,158.752
C01649=1025.431,35.302,-99.020,167.614,47.331,158.752
C01650=1025.425,35.053,-99.004,167.613,47.335,158.752
C01651=1025.419,34.803,-98.988,167.609,47.338,158.753
C01652=1025.413,34.553,-98.972,167.608,47.341,158.753
C01653=1025.406,34.304,-98.956,167.604,47.345,158.753
C01654=1025.401,34.054,-98.941,167.602,47.348,158.754
C01655=1025.394,33.805,-98.925,167.599,47.351,158.754
C01656=1025.388,33.556,-98.909,167.597,47.355,158.754
C01657=1025.383,33.306,-98.893,167.594,47.358,158.754
C01658=1025.376,33.057,-98.878,167.592,47.361,158.755
C01659=1025.370,32.808,-98.861,167.589,47.364,158.755
C01660=1025.364,32.558,-98.846,167.587,47.368,158.755
C01661=1025.358,32.309,-98.830,167.584,47.371,158.756
C01662=1025.352,32.059,-98.815,167.581,47.375,158.756
C01663=1025.345,31.810,-98.799,167.579,47.378,158.756
C01664=1025.339,31.560,-98.783,167.576,47.382,158.757
C01665=1025.334,31.310,-98.767,167.574,47.384,158.757
C01666=1025.328,31.062,-98.752,167.571,47.388,158.757
C01667=1025.322,30.812,-98.736,167.569,47.391,158.757
C01668=1025.316,30.563,-98.720,167.566,47.395,158.758
C01669=1025.309,30.314,-98.705,167.564,47.398,158.758
C01670=1025.304,30.064,-98.689,167.561,47.401,158.758
C01671=1025.297,29.815,-98.673,167.559,47.404,158.759
C01672=1025.291,29.565,-98.658,167.555,47.407,158.759
C01673=1025.285,29.315,-98.642,167.554,47.411,158.759
C01674=1025.279,29.066,-98.627,167.550,47.414,158.759
C01675=1025.273,28.816,-98.610,167.549,47.418,158.760
C01676=1025.268,28.567,-98.595,167.545,47.421,158.760
C01677=1025.261,28.318,-98.579,167.543,47.424,158.760
C01678=1025.256,28.068,-98.564,167.540,47.427,158.760
C01679=1025.250,27.855,-98.551,167.538,47.430,158.761
C01680=1025.245,27.640,-98.537,167.536,47.433,158.761
C01681=1025.240,27.426,-98.524,167.534,47.436,158.761
C01682=1025.234,27.213,-98.511,167.532,47.439,158.761
C01683=1025.229,26.998,-98.497,167.529,47.442,158.762
C01684=1025.223,26.785,-98.484,167.527,47.444,158.762
C01685=1025.219,26.570,-98.471,167.525,47.447,158.762
C01686=1025.214,26.356,-98.457,167.523,47.450,158.762
C01687=1025.207,26.108,-98.442,167.521,47.453,158.763
C01688=1025.201,25.858,-98.427,167.518,47.457,158.763
C01689=1025.195,25.608,-98.411,167.515,47.460,158.763
C01690=1025.189,25.359,-98.396,167.513,47.463,158.764
C01691=1025.183,25.109,-98.380,167.510,47.467,158.764
C01692=1025.177,24.859,-98.365,167.508,47.470,158.764
C01693=1025.170,24.610,-98.350,167.505,47.474,158.765
C01694=1025.165,24.361,-98.334,167.503,47.477,158.765
C01695=1025.159,24.111,-98.319,167.500,47.480,158.765
C01696=1025.153,23.862,-98.303,167.498,47.483,158.765
C01697=1025.146,23.612,-98.288,167.495,47.487,158.766
C01698=1025.140,23.363,-98.273,167.492,47.490,158.766
C01699=1025.132,23.007,-98.252,167.488,47.495,158.766
C01700=1025.123,22.651,-98.230,167.484,47.500,158.767
C01701=1025.114,22.295,-98.207,167.481,47.505,158.767
C01702=1025.105,21.939,-98.186,167.477,47.509,158.768
C01703=1025.100,21.689,-98.170,167.475,47.512,158.768
C01704=1025.093,21.440,-98.155,167.472,47.516,158.768
C01705=1025.087,21.190,-98.140,167.470,47.519,158.768
C01706=1025.081,20.941,-98.124,167.467,47.523,158.769
C01707=1025.075,20.692,-98.110,167.464,47.526,158.769
C01708=1025.070,20.442,-98.094,167.462,47.529,158.769
C01709=1025.063,20.192,-98.079,167.459,47.532,158.769
C01710=1025.056,19.943,-98.063,167.457,47.536,158.770
C01711=1025.051,19.694,-98.048,167.454,47.539,158.770
C01712=1025.045,19.444,-98.033,167.452,47.542,158.770
C01713=1025.039,19.194,-98.018,167.449,47.546,158.771
C01714=1025.032,18.945,-98.003,167.446,47.549,158.771
C01715=1025.027,18.695,-97.988,167.444,47.552,158.771
C01716=1025.021,18.446,-97.973,167.440,47.556,158.771
C01717=1025.014,18.197,-97.958,167.439,47.559,158.772
C01718=1025.008,17.947,-97.943,167.435,47.562,158.772
C01719=1025.003,17.698,-97.927,167.434,47.566,158.772
C01720=1024.996,17.448,-97.912,167.430,47.569,158.773
C01721=1024.990,17.198,-97.898,167.428,47.572,158.773
C01722=1024.984,16.950,-97.883,167.425,47.576,158.773
C01723=1024.978,16.700,-97.868,167.422,47.579,158.773
C01724=1024.972,16.450,-97.852,167.420,47.582,158.774
C01725=1024.966,16.200,-97.838,167.417,47.586,158.774
C01726=1024.960,15.951,-97.823,167.415,47.589,158.774
C01727=1024.954,15.702,-97.808,167.412,47.593,158.775
C01728=1024.947,15.452,-97.793,167.410,47.596,158.775
C01729=1024.942,15.203,-97.778,167.407,47.599,158.775
C01730=1024.936,14.953,-97.763,167.404,47.603,158.775
C01731=1024.929,14.703,-97.748,167.402,47.606,158.776
C01732=1024.924,14.454,-97.733,167.399,47.609,158.776
C01733=1024.917,14.205,-97.718,167.397,47.612,158.776
C01734=1024.912,13.955,-97.703,167.394,47.616,158.776
C01735=1024.906,13.706,-97.688,167.392,47.619,158.777
C01736=1024.899,13.456,-97.673,167.389,47.623,158.777
C01737=1024.893,13.207,-97.658,167.386,47.626,158.777
C01738=1024.887,12.958,-97.644,167.384,47.629,158.778
C01739=1024.881,12.708,-97.629,167.381,47.633,158.778
C01740=1024.874,12.458,-97.614,167.378,47.636,158.778
C01741=1024.869,12.209,-97.599,167.376,47.640,158.778
C01742=1024.863,11.959,-97.585,167.373,47.643,158.779
C01743=1024.856,11.676,-97.569,167.370,47.647,158.779
C01744=1024.848,11.391,-97.552,167.367,47.651,158.779
C01745=1024.842,11.108,-97.535,167.364,47.655,158.780
C01746=1024.834,10.824,-97.519,167.362,47.659,158.780
C01747=1024.828,10.574,-97.504,167.358,47.662,158.780
C01748=1024.822,10.325,-97.489,167.355,47.666,158.781
C01749=1024.816,10.076,-97.474,167.353,47.669,158.781
C01750=1024.810,9.826,-97.459,167.350,47.673,158.781
C01751=1024.804,9.577,-97.446,167.347,47.676,158.781
C01752=1024.797,9.327,-97.431,167.345,47.679,158.782
C01753=1024.791,9.078,-97.417,167.342,47.682,158.782
C01754=1024.785,8.829,-97.402,167.339,47.686,158.782
C01755=1024.779,8.578,-97.387,167.338,47.690,158.783
C01756=1024.773,8.329,-97.373,167.334,47.693,158.783
C01757=1024.767,8.080,-97.358,167.332,47.696,158.783
C01758=1024.761,7.831,-97.343,167.329,47.700,158.783
C01759=1024.755,7.581,-97.329,167.326,47.703,158.784
C01760=1024.748,7.331,-97.314,167.324,47.706,158.784
C01761=1024.743,7.082,-97.300,167.321,47.710,158.784
C01762=1024.736,6.832,-97.285,167.318,47.713,158.784
C01763=1024.731,6.583,-97.271,167.316,47.717,158.785
C01764=1024.724,6.333,-97.256,167.313,47.720,158.785
C01765=1024.718,6.084,-97.243,167.311,47.724,158.785
C01766=1024.712,5.834,-97.228,167.308,47.727,158.786
C01767=1024.706,5.585,-97.213,167.305,47.730,158.786
C01768=1024.700,5.335,-97.199,167.303,47.733,158.786
C01769=1024.694,5.086,-97.184,167.300,47.736,158.786
C01770=1024.688,4.836,-97.169,167.297,47.740,158.787
C01771=1024.682,4.587,-97.155,167.295,47.743,158.787
C01772=1024.676,4.337,-97.140,167.292,47.747,158.787
C01773=1024.670,4.088,-97.126,167.290,47.750,158.787
C01774=1024.663,3.838,-97.112,167.287,47.754,158.788
C01775=1024.657,3.589,-97.098,167.284,47.757,158.788
C01776=1024.651,3.339,-97.083,167.282,47.760,158.788
C01777=1024.646,3.090,-97.069,167.279,47.764,158.788
C01778=1024.639,2.840,-97.054,167.276,47.767,158.789
C01779=1024.634,2.591,-97.040,167.274,47.770,158.789
C01780=1024.627,2.341,-97.025,167.271,47.773,158.789
C01781=1024.622,2.091,-97.011,167.269,47.777,158.790
C01782=1024.615,1.842,-96.996,167.266,47.780,158.790
C01783=1024.609,1.593,-96.983,167.263,47.784,158.790
C01784=1024.603,1.343,-96.968,167.261,47.787,158.790
C01785=1024.597,1.094,-96.953,167.257,47.790,158.790
C01786=1024.592,0.844,-96.940,167.254,47.794,158.791
C01787=1024.585,0.595,-96.925,167.252,47.797,158.791
C01788=1024.580,0.345,-96.911,167.249,47.800,158.791
